LIN {X 0,Y 324.225,Z 783.295,A -85,B 0,C 180,E1 -16076.863,E2 -16076.863} C_VEL
LIN {X 0,Y 323.247,Z 797.636,A -85,B 0,C 180,E1 -16077.399,E2 -16077.399} C_VEL
LIN {X 0,Y 321.791,Z 812,A -85,B 0,C 180,E1 -16078.204,E2 -16078.204} C_VEL
LIN {X 0,Y 320.242,Z 823.952,A -85,B 0,C 180,E1 -16079.097,E2 -16079.097} C_VEL
LIN {X 0,Y 318.471,Z 835.826,A -85,B 0,C 180,E1 -16080.229,E2 -16080.229} C_VEL
LIN {X 0,Y 316.384,Z 847.778,A -85,B 0,C 180,E1 -16081.653,E2 -16081.653} C_VEL
LIN {X 0,Y 314.455,Z 857.682,A -85,B 0,C 180,E1 -16083.091,E2 -16083.091} C_VEL
LIN {X 0,Y 312.599,Z 866.939,A -85,B 0,C 180,E1 -16084.712,E2 -16084.712} C_VEL
LIN {X 0,Y 310.516,Z 876.173,A -85,B 0,C 180,E1 -16086.667,E2 -16086.667} C_VEL
LIN {X 0,Y 308.761,Z 883.843,A -85,B 0,C 180,E1 -16088.642,E2 -16088.642} C_VEL
LIN {X 0,Y 307.38,Z 890.201,A -85,B 0,C 180,E1 -16090.638,E2 -16090.638} C_VEL
LIN {X 0,Y 306.143,Z 895.408,A -85,B 0,C 180,E1 -16092.636,E2 -16092.636} C_VEL
LIN {X 0,Y 305.046,Z 900.883,A -85,B 0,C 180,E1 -16095.319,E2 -16095.319} C_VEL
LIN {X 0,Y 304.213,Z 904.768,A -85,B 0,C 180,E1 -16098,E2 -16098} C_VEL
LIN {X 0,Y 303.829,Z 907.205,A -85,B 0,C 180,E1 -16100.682,E2 -16100.682} C_VEL
LIN {X 0,Y 303.712,Z 908.297,A -85,B 0,C 180,E1 -16103.356,E2 -16103.356} C_VEL
LIN {X 0,Y 303.689,Z 908.077,A -85,B 0,C 180,E1 -16106.019,E2 -16106.019} C_VEL
LIN {X 0,Y 303.703,Z 906.551,A -85,B 0,C 180,E1 -16108.674,E2 -16108.674} C_VEL
LIN {X 0,Y 303.964,Z 903.684,A -85,B 0,C 180,E1 -16111.325,E2 -16111.325} C_VEL
LIN {X 0,Y 304.542,Z 899.397,A -85,B 0,C 180,E1 -16113.97,E2 -16113.97} C_VEL
LIN {X 0,Y 305.582,Z 893.552,A -85,B 0,C 180,E1 -16116.603,E2 -16116.603} C_VEL
LIN {X 0,Y 306.398,Z 887.984,A -85,B 0,C 180,E1 -16118.575,E2 -16118.575} C_VEL
LIN {X 0,Y 307.686,Z 880.207,A -85,B 0,C 180,E1 -16120.828,E2 -16120.828} C_VEL
LIN {X 0,Y 309.255,Z 871.807,A -85,B 0,C 180,E1 -16122.802,E2 -16122.802} C_VEL
LIN {X 0,Y 311.105,Z 861.842,A -85,B 0,C 180,E1 -16124.723,E2 -16124.723} C_VEL
LIN {X 0,Y 312.875,Z 850.729,A -85,B 0,C 180,E1 -16126.475,E2 -16126.475} C_VEL
LIN {X 0,Y 314.508,Z 839.68,A -85,B 0,C 180,E1 -16127.894,E2 -16127.894} C_VEL
LIN {X 0,Y 316.077,Z 827.655,A -85,B 0,C 180,E1 -16129.146,E2 -16129.146} C_VEL
LIN {X 0,Y 317.678,Z 814.307,A -85,B 0,C 180,E1 -16130.223,E2 -16130.223} C_VEL
LIN {X 0,Y 318.794,Z 800.403,A -85,B 0,C 180,E1 -16131.077,E2 -16131.077} C_VEL
LIN {X 0,Y 319.652,Z 785.738,A -85,B 0,C 180,E1 -16131.694,E2 -16131.694} C_VEL
LIN {X 0,Y 320.483,Z 760.014,A -85,B 0,C 180,E1 -16132.31,E2 -16132.31} C_VEL
LIN {X 0,Y 322.515,Z 686.456,A -85,B 0,C 180,E1 -16133.928,E2 -16133.928} C_VEL
LIN {X 0,Y 315.088,Z 668.029,A -85,B 0,C 180,E1 -16135.089,E2 -16135.089} C_VEL
LIN {X 0,Y 307.235,Z 651.005,A -85,B 0,C 180,E1 -16136.326,E2 -16136.326} C_VEL
LIN {X 0,Y 305.705,Z 647.706,A -85,B 0,C 180,E1 -16136.607,E2 -16136.607} C_VEL
LIN {X 0,Y 305.453,Z 646.562,A -85,B 0,C 180,E1 -16137.078,E2 -16137.078} C_VEL
LIN {X 0,Y 305.418,Z 646.57,A -85,B 0,C 180,E1 -16140.414,E2 -16140.414} C_VEL
LIN {X 0,Y 305.462,Z 646.561,A -85,B 0,C 180,E1 -16143.462,E2 -16143.462} C_VEL
LIN {X 0,Y 304.856,Z 646.642,A -85,B 0,C 180,E1 -16144.563,E2 -16144.563} C_VEL
LIN {X 0,Y 301.981,Z 646.998,A -85,B 0,C 180,E1 -16146.353,E2 -16146.353} C_VEL
LIN {X 0,Y 299.499,Z 647.302,A -85,B 0,C 180,E1 -16147.806,E2 -16147.806} C_VEL
LIN {X 0,Y 298.433,Z 647.423,A -85,B 0,C 180,E1 -16148.933,E2 -16148.933} C_VEL
LIN {X 0,Y 298.348,Z 647.43,A -85,B 0,C 180,E1 -16149.315,E2 -16149.315} C_VEL
LIN {X 0,Y 298.402,Z 647.438,A -85,B 0,C 180,E1 -16153.103,E2 -16153.103} C_VEL
LIN {X 0,Y 298.373,Z 647.44,A -85,B 0,C 180,E1 -16156.915,E2 -16156.915} C_VEL
LIN {X 0,Y 298.359,Z 647.429,A -85,B 0,C 180,E1 -16161.017,E2 -16161.017} C_VEL
LIN {X 0,Y 298.406,Z 647.416,A -85,B 0,C 180,E1 -16163.928,E2 -16163.928} C_VEL
LIN {X 0,Y 298.395,Z 647.443,A -85,B 0,C 180,E1 -16167.199,E2 -16167.199} C_VEL
LIN {X 0,Y 298.405,Z 647.428,A -85,B 0,C 180,E1 -16170.625,E2 -16170.625} C_VEL
LIN {X 0,Y 298.442,Z 647.424,A -85,B 0,C 180,E1 -16174.92,E2 -16174.92} C_VEL
LIN {X 0,Y 298.405,Z 647.437,A -85,B 0,C 180,E1 -16177.862,E2 -16177.862} C_VEL
LIN {X 0,Y 298.506,Z 647.422,A -85,B 0,C 180,E1 -16180.754,E2 -16180.754} C_VEL
LIN {X 0,Y 298.588,Z 647.412,A -85,B 0,C 180,E1 -16184.994,E2 -16184.994} C_VEL
LIN {X 0,Y 298.586,Z 647.4,A -85,B 0,C 180,E1 -16189.146,E2 -16189.146} C_VEL
LIN {X 0,Y 298.701,Z 647.398,A -85,B 0,C 180,E1 -16191.884,E2 -16191.884} C_VEL
LIN {X 0,Y 298.639,Z 647.406,A -85,B 0,C 180,E1 -16194.598,E2 -16194.598} C_VEL
LIN {X 0,Y 298.922,Z 647.373,A -85,B 0,C 180,E1 -16198.652,E2 -16198.652} C_VEL
LIN {X 0,Y 298.923,Z 647.365,A -85,B 0,C 180,E1 -16201.347,E2 -16201.347} C_VEL
LIN {X 0,Y 298.788,Z 647.387,A -85,B 0,C 180,E1 -16206.754,E2 -16206.754} C_VEL
LIN {X 0,Y 298.638,Z 647.41,A -85,B 0,C 180,E1 -16209.481,E2 -16209.481} C_VEL
LIN {X 0,Y 298.554,Z 647.42,A -85,B 0,C 180,E1 -16213.615,E2 -16213.615} C_VEL
LIN {X 0,Y 298.551,Z 647.417,A -85,B 0,C 180,E1 -16216.408,E2 -16216.408} C_VEL
LIN {X 0,Y 298.512,Z 647.417,A -85,B 0,C 180,E1 -16219.654,E2 -16219.654} C_VEL
LIN {X 0,Y 298.43,Z 647.428,A -85,B 0,C 180,E1 -16223.6,E2 -16223.6} C_VEL
LIN {X 0,Y 298.491,Z 647.423,A -85,B 0,C 180,E1 -16226.574,E2 -16226.574} C_VEL
LIN {X 0,Y 298.422,Z 647.436,A -85,B 0,C 180,E1 -16229.64,E2 -16229.64} C_VEL
LIN {X 0,Y 298.397,Z 647.439,A -85,B 0,C 180,E1 -16232.8,E2 -16232.8} C_VEL
LIN {X 0,Y 298.467,Z 647.429,A -85,B 0,C 180,E1 -16236.812,E2 -16236.812} C_VEL
LIN {X 0,Y 298.42,Z 647.436,A -85,B 0,C 180,E1 -16241.094,E2 -16241.094} C_VEL
LIN {X 0,Y 298.46,Z 647.431,A -85,B 0,C 180,E1 -16243.115,E2 -16243.115} C_VEL
LIN {X 0,Y 298.403,Z 647.429,A -85,B 0,C 180,E1 -16246.92,E2 -16246.92} C_VEL
LIN {X 0,Y 298.416,Z 647.439,A -85,B 0,C 180,E1 -16251.003,E2 -16251.003} C_VEL
LIN {X 0,Y 298.47,Z 647.46,A -85,B 0,C 180,E1 -16252.143,E2 -16252.143} C_VEL
LIN {X 0,Y 301.205,Z 658.566,A -85,B 0,C 180,E1 -16255.596,E2 -16255.596} C_VEL
LIN {X 0,Y 303.172,Z 667.328,A -85,B 0,C 180,E1 -16258.169,E2 -16258.169} C_VEL
LIN {X 0,Y 310.639,Z 685.569,A -85,B 0,C 180,E1 -16259.416,E2 -16259.416} C_VEL
LIN {X 0,Y 314.632,Z 710.905,A -85,B 0,C 180,E1 -16260.445,E2 -16260.445} C_VEL
LIN {X 0,Y 315.552,Z 718.211,A -85,B 0,C 180,E1 -16260.714,E2 -16260.714} C_VEL
LIN {X 0,Y 313.023,Z 805.174,A -85,B 0,C 180,E1 -16262.686,E2 -16262.686} C_VEL
LIN {X 0,Y 311.976,Z 819.378,A -85,B 0,C 180,E1 -16263.221,E2 -16263.221} C_VEL
LIN {X 0,Y 310.677,Z 833.152,A -85,B 0,C 180,E1 -16264.005,E2 -16264.005} C_VEL
LIN {X 0,Y 309.162,Z 845.617,A -85,B 0,C 180,E1 -16264.951,E2 -16264.951} C_VEL
LIN {X 0,Y 307.467,Z 857.573,A -85,B 0,C 180,E1 -16266.108,E2 -16266.108} C_VEL
LIN {X 0,Y 305.661,Z 869.302,A -85,B 0,C 180,E1 -16267.526,E2 -16267.526} C_VEL
LIN {X 0,Y 303.892,Z 879.332,A -85,B 0,C 180,E1 -16268.994,E2 -16268.994} C_VEL
LIN {X 0,Y 302.222,Z 888.717,A -85,B 0,C 180,E1 -16270.648,E2 -16270.648} C_VEL
LIN {X 0,Y 300.501,Z 898.114,A -85,B 0,C 180,E1 -16272.651,E2 -16272.651} C_VEL
LIN {X 0,Y 299.305,Z 905.27,A -85,B 0,C 180,E1 -16274.493,E2 -16274.493} C_VEL
LIN {X 0,Y 298.259,Z 912.434,A -85,B 0,C 180,E1 -16276.718,E2 -16276.718} C_VEL
LIN {X 0,Y 297.296,Z 918.614,A -85,B 0,C 180,E1 -16279.099,E2 -16279.099} C_VEL
LIN {X 0,Y 296.88,Z 922.825,A -85,B 0,C 180,E1 -16281.148,E2 -16281.148} C_VEL
LIN {X 0,Y 296.684,Z 926.174,A -85,B 0,C 180,E1 -16283.198,E2 -16283.198} C_VEL
LIN {X 0,Y 296.573,Z 929.302,A -85,B 0,C 180,E1 -16285.923,E2 -16285.923} C_VEL
LIN {X 0,Y 296.544,Z 931.034,A -85,B 0,C 180,E1 -16288.642,E2 -16288.642} C_VEL
LIN {X 0,Y 296.581,Z 931.393,A -85,B 0,C 180,E1 -16290,E2 -16290} C_VEL
LIN {X 0,Y 296.545,Z 931.098,A -85,B 0,C 180,E1 -16292.717,E2 -16292.717} C_VEL
LIN {X 0,Y 296.622,Z 929.276,A -85,B 0,C 180,E1 -16295.661,E2 -16295.661} C_VEL
LIN {X 0,Y 296.818,Z 926.457,A -85,B 0,C 180,E1 -16298.167,E2 -16298.167} C_VEL
LIN {X 0,Y 297.389,Z 922.006,A -85,B 0,C 180,E1 -16300.898,E2 -16300.898} C_VEL
LIN {X 0,Y 298.591,Z 915.987,A -85,B 0,C 180,E1 -16303.613,E2 -16303.613} C_VEL
LIN {X 0,Y 300.043,Z 909.183,A -85,B 0,C 180,E1 -16305.991,E2 -16305.991} C_VEL
LIN {X 0,Y 301.762,Z 900.853,A -85,B 0,C 180,E1 -16308.325,E2 -16308.325} C_VEL
LIN {X 0,Y 303.736,Z 892.146,A -85,B 0,C 180,E1 -16310.309,E2 -16310.309} C_VEL
LIN {X 0,Y 306.122,Z 881.619,A -85,B 0,C 180,E1 -16312.26,E2 -16312.26} C_VEL
LIN {X 0,Y 308.672,Z 869.857,A -85,B 0,C 180,E1 -16314.016,E2 -16314.016} C_VEL
LIN {X 0,Y 310.843,Z 858.087,A -85,B 0,C 180,E1 -16315.441,E2 -16315.441} C_VEL
LIN {X 0,Y 312.716,Z 846.881,A -85,B 0,C 180,E1 -16316.53,E2 -16316.53} C_VEL
LIN {X 0,Y 314.636,Z 833.843,A -85,B 0,C 180,E1 -16317.522,E2 -16317.522} C_VEL
LIN {X 0,Y 316.173,Z 821.321,A -85,B 0,C 180,E1 -16318.232,E2 -16318.232} C_VEL
LIN {X 0,Y 317.308,Z 807.323,A -85,B 0,C 180,E1 -16318.799,E2 -16318.799} C_VEL
LIN {X 0,Y 318.368,Z 779.879,A -85,B 0,C 180,E1 -16319.456,E2 -16319.456} C_VEL
LIN {X 0,Y 320.304,Z 717.671,A -85,B 0,C 180,E1 -16320.856,E2 -16320.856} C_VEL
LIN {X 0,Y 316.05,Z 693.353,A -85,B 0,C 180,E1 -16322.001,E2 -16322.001} C_VEL
LIN {X 0,Y 309.511,Z 678.866,A -85,B 0,C 180,E1 -16323.217,E2 -16323.217} C_VEL
LIN {X 0,Y 303.624,Z 666.683,A -85,B 0,C 180,E1 -16324.378,E2 -16324.378} C_VEL
LIN {X 0,Y 301.159,Z 657.209,A -85,B 0,C 180,E1 -16327.492,E2 -16327.492} C_VEL
LIN {X 0,Y 298.416,Z 647.429,A -85,B 0,C 180,E1 -16330.982,E2 -16330.982} C_VEL
LIN {X 0,Y 298.425,Z 647.427,A -85,B 0,C 180,E1 -16333.109,E2 -16333.109} C_VEL
LIN {X 0,Y 298.431,Z 647.424,A -85,B 0,C 180,E1 -16336.926,E2 -16336.926} C_VEL
LIN {X 0,Y 298.425,Z 647.431,A -85,B 0,C 180,E1 -16341.001,E2 -16341.001} C_VEL
LIN {X 0,Y 298.432,Z 647.421,A -85,B 0,C 180,E1 -16343.932,E2 -16343.932} C_VEL
LIN {X 0,Y 298.395,Z 647.411,A -85,B 0,C 180,E1 -16347.983,E2 -16347.983} C_VEL
LIN {X 0,Y 298.464,Z 647.432,A -85,B 0,C 180,E1 -16351.905,E2 -16351.905} C_VEL
LIN {X 0,Y 298.486,Z 647.425,A -85,B 0,C 180,E1 -16354.924,E2 -16354.924} C_VEL
LIN {X 0,Y 298.451,Z 647.432,A -85,B 0,C 180,E1 -16359.316,E2 -16359.316} C_VEL
LIN {X 0,Y 298.539,Z 647.414,A -85,B 0,C 180,E1 -16362.18,E2 -16362.18} C_VEL
LIN {X 0,Y 298.594,Z 647.412,A -85,B 0,C 180,E1 -16364.995,E2 -16364.995} C_VEL
LIN {X 0,Y 298.593,Z 647.414,A -85,B 0,C 180,E1 -16369.147,E2 -16369.147} C_VEL
LIN {X 0,Y 298.742,Z 647.389,A -85,B 0,C 180,E1 -16371.886,E2 -16371.886} C_VEL
LIN {X 0,Y 298.658,Z 647.401,A -85,B 0,C 180,E1 -16374.599,E2 -16374.599} C_VEL
LIN {X 0,Y 298.923,Z 647.374,A -85,B 0,C 180,E1 -16378.653,E2 -16378.653} C_VEL
LIN {X 0,Y 298.923,Z 647.366,A -85,B 0,C 180,E1 -16381.348,E2 -16381.348} C_VEL
LIN {X 0,Y 298.789,Z 647.386,A -85,B 0,C 180,E1 -16386.755,E2 -16386.755} C_VEL
LIN {X 0,Y 298.637,Z 647.405,A -85,B 0,C 180,E1 -16389.482,E2 -16389.482} C_VEL
LIN {X 0,Y 298.554,Z 647.418,A -85,B 0,C 180,E1 -16393.616,E2 -16393.616} C_VEL
LIN {X 0,Y 298.551,Z 647.417,A -85,B 0,C 180,E1 -16396.409,E2 -16396.409} C_VEL
LIN {X 0,Y 298.499,Z 647.418,A -85,B 0,C 180,E1 -16399.648,E2 -16399.648} C_VEL
LIN {X 0,Y 298.425,Z 647.427,A -85,B 0,C 180,E1 -16403.601,E2 -16403.601} C_VEL
LIN {X 0,Y 298.414,Z 647.433,A -85,B 0,C 180,E1 -16406.582,E2 -16406.582} C_VEL
LIN {X 0,Y 298.399,Z 647.411,A -85,B 0,C 180,E1 -16409.644,E2 -16409.644} C_VEL
LIN {X 0,Y 298.394,Z 647.442,A -85,B 0,C 180,E1 -16412.801,E2 -16412.801} C_VEL
LIN {X 0,Y 298.43,Z 647.432,A -85,B 0,C 180,E1 -16416.803,E2 -16416.803} C_VEL
LIN {X 0,Y 298.375,Z 647.435,A -85,B 0,C 180,E1 -16419.492,E2 -16419.492} C_VEL
LIN {X 0,Y 298.401,Z 647.443,A -85,B 0,C 180,E1 -16423.104,E2 -16423.104} C_VEL
LIN {X 0,Y 298.373,Z 647.445,A -85,B 0,C 180,E1 -16426.915,E2 -16426.915} C_VEL
LIN {X 0,Y 298.393,Z 647.622,A -85,B 0,C 180,E1 -16429.581,E2 -16429.581} C_VEL
LIN {X 0,Y 298.698,Z 648.824,A -85,B 0,C 180,E1 -16430.006,E2 -16430.006} C_VEL
LIN {X 0,Y 308.386,Z 665.956,A -85,B 0,C 180,E1 -16431.853,E2 -16431.853} C_VEL
LIN {X 0,Y 316.216,Z 681.809,A -85,B 0,C 180,E1 -16433.288,E2 -16433.288} C_VEL
LIN {X 0,Y 321.076,Z 692.716,A -85,B 0,C 180,E1 -16434.159,E2 -16434.159} C_VEL
LIN {X 0,Y 318.105,Z 784.085,A -85,B 0,C 180,E1 -16436.235,E2 -16436.235} C_VEL
LIN {X 0,Y 317.087,Z 798.194,A -85,B 0,C 180,E1 -16436.779,E2 -16436.779} C_VEL
LIN {X 0,Y 315.58,Z 812.483,A -85,B 0,C 180,E1 -16437.597,E2 -16437.597} C_VEL
LIN {X 0,Y 313.967,Z 824.361,A -85,B 0,C 180,E1 -16438.501,E2 -16438.501} C_VEL
LIN {X 0,Y 311.997,Z 836.946,A -85,B 0,C 180,E1 -16439.734,E2 -16439.734} C_VEL
LIN {X 0,Y 309.843,Z 848.746,A -85,B 0,C 180,E1 -16441.184,E2 -16441.184} C_VEL
LIN {X 0,Y 307.635,Z 859.512,A -85,B 0,C 180,E1 -16442.812,E2 -16442.812} C_VEL
LIN {X 0,Y 305.341,Z 870.141,A -85,B 0,C 180,E1 -16444.798,E2 -16444.798} C_VEL
LIN {X 0,Y 303.243,Z 878.881,A -85,B 0,C 180,E1 -16446.797,E2 -16446.797} C_VEL
LIN {X 0,Y 301.287,Z 886.951,A -85,B 0,C 180,E1 -16449.07,E2 -16449.07} C_VEL
LIN {X 0,Y 299.673,Z 893.906,A -85,B 0,C 180,E1 -16451.542,E2 -16451.542} C_VEL
LIN {X 0,Y 298.323,Z 899.794,A -85,B 0,C 180,E1 -16454.281,E2 -16454.281} C_VEL
LIN {X 0,Y 297.578,Z 903.189,A -85,B 0,C 180,E1 -16456.339,E2 -16456.339} C_VEL
LIN {X 0,Y 296.9,Z 906.377,A -85,B 0,C 180,E1 -16459.084,E2 -16459.084} C_VEL
LIN {X 0,Y 296.682,Z 908.165,A -85,B 0,C 180,E1 -16461.829,E2 -16461.829} C_VEL
LIN {X 0,Y 296.623,Z 908.631,A -85,B 0,C 180,E1 -16464.562,E2 -16464.562} C_VEL
LIN {X 0,Y 296.604,Z 907.792,A -85,B 0,C 180,E1 -16467.284,E2 -16467.284} C_VEL
LIN {X 0,Y 296.718,Z 905.636,A -85,B 0,C 180,E1 -16470,E2 -16470} C_VEL
LIN {X 0,Y 297.101,Z 902.109,A -85,B 0,C 180,E1 -16472.712,E2 -16472.712} C_VEL
LIN {X 0,Y 297.822,Z 898.501,A -85,B 0,C 180,E1 -16474.738,E2 -16474.738} C_VEL
LIN {X 0,Y 298.818,Z 892.248,A -85,B 0,C 180,E1 -16477.433,E2 -16477.433} C_VEL
LIN {X 0,Y 299.862,Z 886.39,A -85,B 0,C 180,E1 -16479.443,E2 -16479.443} C_VEL
LIN {X 0,Y 301.192,Z 878.162,A -85,B 0,C 180,E1 -16481.747,E2 -16481.747} C_VEL
LIN {X 0,Y 302.992,Z 869.277,A -85,B 0,C 180,E1 -16483.754,E2 -16483.754} C_VEL
LIN {X 0,Y 304.932,Z 858.691,A -85,B 0,C 180,E1 -16485.713,E2 -16485.713} C_VEL
LIN {X 0,Y 306.708,Z 847.993,A -85,B 0,C 180,E1 -16487.331,E2 -16487.331} C_VEL
LIN {X 0,Y 308.334,Z 836.313,A -85,B 0,C 180,E1 -16488.782,E2 -16488.782} C_VEL
LIN {X 0,Y 310.134,Z 823.398,A -85,B 0,C 180,E1 -16490.045,E2 -16490.045} C_VEL
LIN {X 0,Y 311.63,Z 809.884,A -85,B 0,C 180,E1 -16491.065,E2 -16491.065} C_VEL
LIN {X 0,Y 312.735,Z 795.632,A -85,B 0,C 180,E1 -16491.852,E2 -16491.852} C_VEL
LIN {X 0,Y 313.458,Z 781.713,A -85,B 0,C 180,E1 -16492.362,E2 -16492.362} C_VEL
LIN {X 0,Y 316.225,Z 688.388,A -85,B 0,C 180,E1 -16494.465,E2 -16494.465} C_VEL
LIN {X 0,Y 308.861,Z 670.042,A -85,B 0,C 180,E1 -16495.659,E2 -16495.659} C_VEL
LIN {X 0,Y 300.183,Z 651.551,A -85,B 0,C 180,E1 -16497.075,E2 -16497.075} C_VEL
LIN {X 0,Y 298.544,Z 648.169,A -85,B 0,C 180,E1 -16497.351,E2 -16497.351} C_VEL
LIN {X 0,Y 298.402,Z 647.444,A -85,B 0,C 180,E1 -16497.637,E2 -16497.637} C_VEL
LIN {X 0,Y 298.39,Z 647.443,A -85,B 0,C 180,E1 -16502.014,E2 -16502.014} C_VEL
LIN {X 0,Y 298.432,Z 647.435,A -85,B 0,C 180,E1 -16504.487,E2 -16504.487} C_VEL
LIN {X 0,Y 298.389,Z 647.441,A -85,B 0,C 180,E1 -16507.762,E2 -16507.762} C_VEL
LIN {X 0,Y 298.348,Z 647.43,A -85,B 0,C 180,E1 -16509.315,E2 -16509.315} C_VEL
LIN {X 0,Y 297.68,Z 647.514,A -85,B 0,C 180,E1 -16510.442,E2 -16510.442} C_VEL
LIN {X 0,Y 294.805,Z 647.887,A -85,B 0,C 180,E1 -16512.276,E2 -16512.276} C_VEL
LIN {X 0,Y 292.376,Z 648.187,A -85,B 0,C 180,E1 -16513.765,E2 -16513.765} C_VEL
LIN {X 0,Y 291.35,Z 648.316,A -85,B 0,C 180,E1 -16514.919,E2 -16514.919} C_VEL
LIN {X 0,Y 291.275,Z 648.325,A -85,B 0,C 180,E1 -16515.309,E2 -16515.309} C_VEL
LIN {X 0,Y 291.297,Z 648.324,A -85,B 0,C 180,E1 -16519.351,E2 -16519.351} C_VEL
LIN {X 0,Y 291.389,Z 648.282,A -85,B 0,C 180,E1 -16522.916,E2 -16522.916} C_VEL
LIN {X 0,Y 291.346,Z 648.316,A -85,B 0,C 180,E1 -16526.301,E2 -16526.301} C_VEL
LIN {X 0,Y 291.368,Z 648.303,A -85,B 0,C 180,E1 -16530.268,E2 -16530.268} C_VEL
LIN {X 0,Y 291.361,Z 648.311,A -85,B 0,C 180,E1 -16534.266,E2 -16534.266} C_VEL
LIN {X 0,Y 291.367,Z 648.306,A -85,B 0,C 180,E1 -16537.298,E2 -16537.298} C_VEL
LIN {X 0,Y 291.442,Z 648.302,A -85,B 0,C 180,E1 -16540.269,E2 -16540.269} C_VEL
LIN {X 0,Y 291.517,Z 648.292,A -85,B 0,C 180,E1 -16544.653,E2 -16544.653} C_VEL
LIN {X 0,Y 291.532,Z 648.279,A -85,B 0,C 180,E1 -16548.88,E2 -16548.88} C_VEL
LIN {X 0,Y 291.654,Z 648.273,A -85,B 0,C 180,E1 -16551.686,E2 -16551.686} C_VEL
LIN {X 0,Y 291.608,Z 648.282,A -85,B 0,C 180,E1 -16554.467,E2 -16554.467} C_VEL
LIN {X 0,Y 291.889,Z 648.249,A -85,B 0,C 180,E1 -16558.62,E2 -16558.62} C_VEL
LIN {X 0,Y 291.889,Z 648.241,A -85,B 0,C 180,E1 -16561.379,E2 -16561.379} C_VEL
LIN {X 0,Y 291.737,Z 648.265,A -85,B 0,C 180,E1 -16566.918,E2 -16566.918} C_VEL
LIN {X 0,Y 291.577,Z 648.286,A -85,B 0,C 180,E1 -16569.713,E2 -16569.713} C_VEL
LIN {X 0,Y 291.524,Z 648.294,A -85,B 0,C 180,E1 -16573.95,E2 -16573.95} C_VEL
LIN {X 0,Y 291.489,Z 648.297,A -85,B 0,C 180,E1 -16576.817,E2 -16576.817} C_VEL
LIN {X 0,Y 291.452,Z 648.297,A -85,B 0,C 180,E1 -16579.874,E2 -16579.874} C_VEL
LIN {X 0,Y 291.384,Z 648.307,A -85,B 0,C 180,E1 -16584.206,E2 -16584.206} C_VEL
LIN {X 0,Y 291.424,Z 648.301,A -85,B 0,C 180,E1 -16587.271,E2 -16587.271} C_VEL
LIN {X 0,Y 291.339,Z 648.315,A -85,B 0,C 180,E1 -16590.436,E2 -16590.436} C_VEL
LIN {X 0,Y 291.346,Z 648.316,A -85,B 0,C 180,E1 -16593.698,E2 -16593.698} C_VEL
LIN {X 0,Y 291.402,Z 648.31,A -85,B 0,C 180,E1 -16597.26,E2 -16597.26} C_VEL
LIN {X 0,Y 291.379,Z 648.316,A -85,B 0,C 180,E1 -16600.634,E2 -16600.634} C_VEL
LIN {X 0,Y 291.333,Z 648.318,A -85,B 0,C 180,E1 -16604.393,E2 -16604.393} C_VEL
LIN {X 0,Y 291.328,Z 648.321,A -85,B 0,C 180,E1 -16608.404,E2 -16608.404} C_VEL
LIN {X 0,Y 291.439,Z 648.509,A -85,B 0,C 180,E1 -16611.543,E2 -16611.543} C_VEL
LIN {X 0,Y 294.13,Z 659.279,A -85,B 0,C 180,E1 -16615.008,E2 -16615.008} C_VEL
LIN {X 0,Y 295.851,Z 666.97,A -85,B 0,C 180,E1 -16617.347,E2 -16617.347} C_VEL
LIN {X 0,Y 304.416,Z 687.348,A -85,B 0,C 180,E1 -16618.832,E2 -16618.832} C_VEL
LIN {X 0,Y 307.154,Z 703.717,A -85,B 0,C 180,E1 -16619.539,E2 -16619.539} C_VEL
LIN {X 0,Y 309.223,Z 719.038,A -85,B 0,C 180,E1 -16620.138,E2 -16620.138} C_VEL
LIN {X 0,Y 306.575,Z 805.95,A -85,B 0,C 180,E1 -16622.155,E2 -16622.155} C_VEL
LIN {X 0,Y 305.41,Z 820.519,A -85,B 0,C 180,E1 -16622.737,E2 -16622.737} C_VEL
LIN {X 0,Y 304.155,Z 833.362,A -85,B 0,C 180,E1 -16623.497,E2 -16623.497} C_VEL
LIN {X 0,Y 302.452,Z 846.611,A -85,B 0,C 180,E1 -16624.54,E2 -16624.54} C_VEL
LIN {X 0,Y 300.52,Z 859.533,A -85,B 0,C 180,E1 -16625.858,E2 -16625.858} C_VEL
LIN {X 0,Y 298.669,Z 871.063,A -85,B 0,C 180,E1 -16627.336,E2 -16627.336} C_VEL
LIN {X 0,Y 296.806,Z 880.745,A -85,B 0,C 180,E1 -16628.832,E2 -16628.832} C_VEL
LIN {X 0,Y 294.836,Z 891.508,A -85,B 0,C 180,E1 -16630.867,E2 -16630.867} C_VEL
LIN {X 0,Y 293.14,Z 900.385,A -85,B 0,C 180,E1 -16632.921,E2 -16632.921} C_VEL
LIN {X 0,Y 292.024,Z 907.781,A -85,B 0,C 180,E1 -16635.006,E2 -16635.006} C_VEL
LIN {X 0,Y 290.821,Z 914.841,A -85,B 0,C 180,E1 -16637.438,E2 -16637.438} C_VEL
LIN {X 0,Y 290.094,Z 919.733,A -85,B 0,C 180,E1 -16639.531,E2 -16639.531} C_VEL
LIN {X 0,Y 289.654,Z 924.792,A -85,B 0,C 180,E1 -16642.331,E2 -16642.331} C_VEL
LIN {X 0,Y 289.515,Z 927.59,A -85,B 0,C 180,E1 -16644.428,E2 -16644.428} C_VEL
LIN {X 0,Y 289.486,Z 930.038,A -85,B 0,C 180,E1 -16647.217,E2 -16647.217} C_VEL
LIN {X 0,Y 289.496,Z 931.115,A -85,B 0,C 180,E1 -16650,E2 -16650} C_VEL
LIN {X 0,Y 289.471,Z 930.842,A -85,B 0,C 180,E1 -16652.783,E2 -16652.783} C_VEL
LIN {X 0,Y 289.515,Z 929.228,A -85,B 0,C 180,E1 -16655.572,E2 -16655.572} C_VEL
LIN {X 0,Y 289.754,Z 926.246,A -85,B 0,C 180,E1 -16658.368,E2 -16658.368} C_VEL
LIN {X 0,Y 290.357,Z 921.819,A -85,B 0,C 180,E1 -16661.165,E2 -16661.165} C_VEL
LIN {X 0,Y 291.637,Z 915.832,A -85,B 0,C 180,E1 -16663.945,E2 -16663.945} C_VEL
LIN {X 0,Y 293.185,Z 908.693,A -85,B 0,C 180,E1 -16666.495,E2 -16666.495} C_VEL
LIN {X 0,Y 294.988,Z 900.771,A -85,B 0,C 180,E1 -16668.762,E2 -16668.762} C_VEL
LIN {X 0,Y 297.056,Z 892.106,A -85,B 0,C 180,E1 -16670.786,E2 -16670.786} C_VEL
LIN {X 0,Y 299.564,Z 881.627,A -85,B 0,C 180,E1 -16672.774,E2 -16672.774} C_VEL
LIN {X 0,Y 302.186,Z 869.924,A -85,B 0,C 180,E1 -16674.565,E2 -16674.565} C_VEL
LIN {X 0,Y 304.452,Z 858.227,A -85,B 0,C 180,E1 -16676.014,E2 -16676.014} C_VEL
LIN {X 0,Y 306.677,Z 845.358,A -85,B 0,C 180,E1 -16677.279,E2 -16677.279} C_VEL
LIN {X 0,Y 308.729,Z 831.97,A -85,B 0,C 180,E1 -16678.28,E2 -16678.28} C_VEL
LIN {X 0,Y 310.214,Z 819.654,A -85,B 0,C 180,E1 -16678.964,E2 -16678.964} C_VEL
LIN {X 0,Y 311.332,Z 806.097,A -85,B 0,C 180,E1 -16679.498,E2 -16679.498} C_VEL
LIN {X 0,Y 313.639,Z 740.667,A -85,B 0,C 180,E1 -16681.023,E2 -16681.023} C_VEL
LIN {X 0,Y 314.282,Z 718.374,A -85,B 0,C 180,E1 -16681.543,E2 -16681.543} C_VEL
LIN {X 0,Y 310.455,Z 696.266,A -85,B 0,C 180,E1 -16682.615,E2 -16682.615} C_VEL
LIN {X 0,Y 304.115,Z 682.195,A -85,B 0,C 180,E1 -16683.839,E2 -16683.839} C_VEL
LIN {X 0,Y 296.363,Z 666.32,A -85,B 0,C 180,E1 -16685.429,E2 -16685.429} C_VEL
LIN {X 0,Y 293.326,Z 655.076,A -85,B 0,C 180,E1 -16689.327,E2 -16689.327} C_VEL
LIN {X 0,Y 291.359,Z 648.316,A -85,B 0,C 180,E1 -16691.854,E2 -16691.854} C_VEL
LIN {X 0,Y 291.323,Z 648.322,A -85,B 0,C 180,E1 -16695.605,E2 -16695.605} C_VEL
LIN {X 0,Y 291.376,Z 648.309,A -85,B 0,C 180,E1 -16699.365,E2 -16699.365} C_VEL
LIN {X 0,Y 291.428,Z 648.286,A -85,B 0,C 180,E1 -16702.923,E2 -16702.923} C_VEL
LIN {X 0,Y 291.345,Z 648.314,A -85,B 0,C 180,E1 -16706.302,E2 -16706.302} C_VEL
LIN {X 0,Y 291.387,Z 648.296,A -85,B 0,C 180,E1 -16710.26,E2 -16710.26} C_VEL
LIN {X 0,Y 291.417,Z 648.302,A -85,B 0,C 180,E1 -16714.272,E2 -16714.272} C_VEL
LIN {X 0,Y 291.382,Z 648.305,A -85,B 0,C 180,E1 -16717.3,E2 -16717.3} C_VEL
LIN {X 0,Y 291.459,Z 648.302,A -85,B 0,C 180,E1 -16720.271,E2 -16720.271} C_VEL
LIN {X 0,Y 291.556,Z 648.29,A -85,B 0,C 180,E1 -16724.624,E2 -16724.624} C_VEL
LIN {X 0,Y 291.537,Z 648.294,A -85,B 0,C 180,E1 -16728.881,E2 -16728.881} C_VEL
LIN {X 0,Y 291.688,Z 648.266,A -85,B 0,C 180,E1 -16731.688,E2 -16731.688} C_VEL
LIN {X 0,Y 291.628,Z 648.277,A -85,B 0,C 180,E1 -16734.469,E2 -16734.469} C_VEL
LIN {X 0,Y 291.89,Z 648.25,A -85,B 0,C 180,E1 -16738.621,E2 -16738.621} C_VEL
LIN {X 0,Y 291.89,Z 648.242,A -85,B 0,C 180,E1 -16741.38,E2 -16741.38} C_VEL
LIN {X 0,Y 291.737,Z 648.266,A -85,B 0,C 180,E1 -16746.919,E2 -16746.919} C_VEL
LIN {X 0,Y 291.577,Z 648.282,A -85,B 0,C 180,E1 -16749.714,E2 -16749.714} C_VEL
LIN {X 0,Y 291.524,Z 648.293,A -85,B 0,C 180,E1 -16753.951,E2 -16753.951} C_VEL
LIN {X 0,Y 291.488,Z 648.301,A -85,B 0,C 180,E1 -16756.818,E2 -16756.818} C_VEL
LIN {X 0,Y 291.452,Z 648.296,A -85,B 0,C 180,E1 -16759.875,E2 -16759.875} C_VEL
LIN {X 0,Y 291.366,Z 648.309,A -85,B 0,C 180,E1 -16764.209,E2 -16764.209} C_VEL
LIN {X 0,Y 291.36,Z 648.303,A -85,B 0,C 180,E1 -16767.278,E2 -16767.278} C_VEL
LIN {X 0,Y 291.322,Z 648.3,A -85,B 0,C 180,E1 -16770.439,E2 -16770.439} C_VEL
LIN {X 0,Y 291.345,Z 648.312,A -85,B 0,C 180,E1 -16773.699,E2 -16773.699} C_VEL
LIN {X 0,Y 291.361,Z 648.313,A -85,B 0,C 180,E1 -16777.25,E2 -16777.25} C_VEL
LIN {X 0,Y 291.301,Z 648.305,A -85,B 0,C 180,E1 -16780.649,E2 -16780.649} C_VEL
LIN {X 0,Y 291.292,Z 648.319,A -85,B 0,C 180,E1 -16784.402,E2 -16784.402} C_VEL
LIN {X 0,Y 291.326,Z 648.339,A -85,B 0,C 180,E1 -16788.642,E2 -16788.642} C_VEL
LIN {X 0,Y 291.428,Z 649.017,A -85,B 0,C 180,E1 -16788.904,E2 -16788.904} C_VEL
LIN {X 0,Y 292.744,Z 651.781,A -85,B 0,C 180,E1 -16789.198,E2 -16789.198} C_VEL
LIN {X 0,Y 294.482,Z 654.35,A -85,B 0,C 180,E1 -16789.543,E2 -16789.543} C_VEL
LIN {X 0,Y 301.594,Z 666.811,A -85,B 0,C 180,E1 -16790.95,E2 -16790.95} C_VEL
LIN {X 0,Y 308.318,Z 679.777,A -85,B 0,C 180,E1 -16792.231,E2 -16792.231} C_VEL
LIN {X 0,Y 315.092,Z 694.702,A -85,B 0,C 180,E1 -16793.497,E2 -16793.497} C_VEL
LIN {X 0,Y 312,Z 785.032,A -85,B 0,C 180,E1 -16795.59,E2 -16795.59} C_VEL
LIN {X 0,Y 310.88,Z 799.519,A -85,B 0,C 180,E1 -16796.173,E2 -16796.173} C_VEL
LIN {X 0,Y 309.417,Z 812.968,A -85,B 0,C 180,E1 -16796.967,E2 -16796.967} C_VEL
LIN {X 0,Y 307.877,Z 823.87,A -85,B 0,C 180,E1 -16797.799,E2 -16797.799} C_VEL
LIN {X 0,Y 305.819,Z 836.634,A -85,B 0,C 180,E1 -16799.056,E2 -16799.056} C_VEL
LIN {X 0,Y 303.556,Z 848.538,A -85,B 0,C 180,E1 -16800.529,E2 -16800.529} C_VEL
LIN {X 0,Y 301.246,Z 859.385,A -85,B 0,C 180,E1 -16802.187,E2 -16802.187} C_VEL
LIN {X 0,Y 298.849,Z 870.082,A -85,B 0,C 180,E1 -16804.211,E2 -16804.211} C_VEL
LIN {X 0,Y 296.653,Z 878.876,A -85,B 0,C 180,E1 -16806.25,E2 -16806.25} C_VEL
LIN {X 0,Y 294.677,Z 886.633,A -85,B 0,C 180,E1 -16808.459,E2 -16808.459} C_VEL
LIN {X 0,Y 292.836,Z 894.006,A -85,B 0,C 180,E1 -16811.095,E2 -16811.095} C_VEL
LIN {X 0,Y 291.391,Z 899.941,A -85,B 0,C 180,E1 -16813.897,E2 -16813.897} C_VEL
LIN {X 0,Y 290.605,Z 903.355,A -85,B 0,C 180,E1 -16816.005,E2 -16816.005} C_VEL
LIN {X 0,Y 289.854,Z 906.591,A -85,B 0,C 180,E1 -16818.815,E2 -16818.815} C_VEL
LIN {X 0,Y 289.616,Z 908.415,A -85,B 0,C 180,E1 -16821.628,E2 -16821.628} C_VEL
LIN {X 0,Y 289.559,Z 908.912,A -85,B 0,C 180,E1 -16824.429,E2 -16824.429} C_VEL
LIN {X 0,Y 289.528,Z 908.106,A -85,B 0,C 180,E1 -16827.217,E2 -16827.217} C_VEL
LIN {X 0,Y 289.626,Z 905.984,A -85,B 0,C 180,E1 -16830,E2 -16830} C_VEL
LIN {X 0,Y 290.02,Z 902.491,A -85,B 0,C 180,E1 -16832.778,E2 -16832.778} C_VEL
LIN {X 0,Y 290.767,Z 898.92,A -85,B 0,C 180,E1 -16834.853,E2 -16834.853} C_VEL
LIN {X 0,Y 291.788,Z 892.707,A -85,B 0,C 180,E1 -16837.613,E2 -16837.613} C_VEL
LIN {X 0,Y 293.074,Z 885.7,A -85,B 0,C 180,E1 -16840.041,E2 -16840.041} C_VEL
LIN {X 0,Y 294.524,Z 877.243,A -85,B 0,C 180,E1 -16842.402,E2 -16842.402} C_VEL
LIN {X 0,Y 296.454,Z 868.272,A -85,B 0,C 180,E1 -16844.414,E2 -16844.414} C_VEL
LIN {X 0,Y 298.528,Z 857.428,A -85,B 0,C 180,E1 -16846.41,E2 -16846.41} C_VEL
LIN {X 0,Y 300.424,Z 846.408,A -85,B 0,C 180,E1 -16848.057,E2 -16848.057} C_VEL
LIN {X 0,Y 302.14,Z 834.27,A -85,B 0,C 180,E1 -16849.535,E2 -16849.535} C_VEL
LIN {X 0,Y 303.773,Z 822.598,A -85,B 0,C 180,E1 -16850.66,E2 -16850.66} C_VEL
LIN {X 0,Y 305.277,Z 808.644,A -85,B 0,C 180,E1 -16851.703,E2 -16851.703} C_VEL
LIN {X 0,Y 306.37,Z 794.668,A -85,B 0,C 180,E1 -16852.463,E2 -16852.463} C_VEL
LIN {X 0,Y 307.138,Z 780.5,A -85,B 0,C 180,E1 -16852.965,E2 -16852.965} C_VEL
LIN {X 0,Y 309.867,Z 690.077,A -85,B 0,C 180,E1 -16855.039,E2 -16855.039} C_VEL
LIN {X 0,Y 303.079,Z 673.187,A -85,B 0,C 180,E1 -16856.178,E2 -16856.178} C_VEL
LIN {X 0,Y 295.601,Z 657.05,A -85,B 0,C 180,E1 -16857.441,E2 -16857.441} C_VEL
LIN {X 0,Y 292.562,Z 651.486,A -85,B 0,C 180,E1 -16857.949,E2 -16857.949} C_VEL
LIN {X 0,Y 291.451,Z 648.879,A -85,B 0,C 180,E1 -16858.154,E2 -16858.154} C_VEL
LIN {X 0,Y 291.351,Z 648.317,A -85,B 0,C 180,E1 -16858.251,E2 -16858.251} C_VEL
LIN {X 0,Y 291.34,Z 648.32,A -85,B 0,C 180,E1 -16862.401,E2 -16862.401} C_VEL
LIN {X 0,Y 291.358,Z 648.318,A -85,B 0,C 180,E1 -16865.375,E2 -16865.375} C_VEL
LIN {X 0,Y 291.307,Z 648.311,A -85,B 0,C 180,E1 -16868.849,E2 -16868.849} C_VEL
LIN {X 0,Y 291.316,Z 648.323,A -85,B 0,C 180,E1 -16872.493,E2 -16872.493} C_VEL
LIN {X 0,Y 291.275,Z 648.325,A -85,B 0,C 180,E1 -16875.309,E2 -16875.309} C_VEL
LIN {X 0,Y 290.621,Z 648.412,A -85,B 0,C 180,E1 -16876.462,E2 -16876.462} C_VEL
LIN {X 0,Y 287.745,Z 648.766,A -85,B 0,C 180,E1 -16878.339,E2 -16878.339} C_VEL
LIN {X 0,Y 285.317,Z 649.066,A -85,B 0,C 180,E1 -16879.862,E2 -16879.862} C_VEL
LIN {X 0,Y 284.307,Z 649.177,A -85,B 0,C 180,E1 -16881.044,E2 -16881.044} C_VEL
LIN {X 0,Y 284.243,Z 649.178,A -85,B 0,C 180,E1 -16881.444,E2 -16881.444} C_VEL
LIN {X 0,Y 284.339,Z 649.176,A -85,B 0,C 180,E1 -16884.653,E2 -16884.653} C_VEL
LIN {X 0,Y 284.288,Z 649.19,A -85,B 0,C 180,E1 -16888.724,E2 -16888.724} C_VEL
LIN {X 0,Y 284.286,Z 649.197,A -85,B 0,C 180,E1 -16891.984,E2 -16891.984} C_VEL
LIN {X 0,Y 284.323,Z 649.177,A -85,B 0,C 180,E1 -16896.147,E2 -16896.147} C_VEL
LIN {X 0,Y 284.379,Z 649.183,A -85,B 0,C 180,E1 -16899.904,E2 -16899.904} C_VEL
LIN {X 0,Y 284.457,Z 649.171,A -85,B 0,C 180,E1 -16904.486,E2 -16904.486} C_VEL
LIN {X 0,Y 284.485,Z 649.159,A -85,B 0,C 180,E1 -16908.601,E2 -16908.601} C_VEL
LIN {X 0,Y 284.611,Z 649.148,A -85,B 0,C 180,E1 -16911.479,E2 -16911.479} C_VEL
LIN {X 0,Y 284.577,Z 649.158,A -85,B 0,C 180,E1 -16914.33,E2 -16914.33} C_VEL
LIN {X 0,Y 284.855,Z 649.126,A -85,B 0,C 180,E1 -16918.586,E2 -16918.586} C_VEL
LIN {X 0,Y 284.856,Z 649.118,A -85,B 0,C 180,E1 -16921.413,E2 -16921.413} C_VEL
LIN {X 0,Y 284.688,Z 649.143,A -85,B 0,C 180,E1 -16927.09,E2 -16927.09} C_VEL
LIN {X 0,Y 284.521,Z 649.162,A -85,B 0,C 180,E1 -16929.957,E2 -16929.957} C_VEL
LIN {X 0,Y 284.484,Z 649.167,A -85,B 0,C 180,E1 -16934.302,E2 -16934.302} C_VEL
LIN {X 0,Y 284.428,Z 649.177,A -85,B 0,C 180,E1 -16937.248,E2 -16937.248} C_VEL
LIN {X 0,Y 284.379,Z 649.179,A -85,B 0,C 180,E1 -16940.242,E2 -16940.242} C_VEL
LIN {X 0,Y 284.34,Z 649.189,A -85,B 0,C 180,E1 -16944.846,E2 -16944.846} C_VEL
LIN {X 0,Y 284.333,Z 649.186,A -85,B 0,C 180,E1 -16948.01,E2 -16948.01} C_VEL
LIN {X 0,Y 284.298,Z 649.192,A -85,B 0,C 180,E1 -16951.274,E2 -16951.274} C_VEL
LIN {X 0,Y 284.363,Z 649.188,A -85,B 0,C 180,E1 -16955.354,E2 -16955.354} C_VEL
LIN {X 0,Y 284.334,Z 649.193,A -85,B 0,C 180,E1 -16958.165,E2 -16958.165} C_VEL
LIN {X 0,Y 284.304,Z 649.193,A -85,B 0,C 180,E1 -16961.87,E2 -16961.87} C_VEL
LIN {X 0,Y 284.266,Z 649.195,A -85,B 0,C 180,E1 -16965.805,E2 -16965.805} C_VEL
LIN {X 0,Y 284.307,Z 649.197,A -85,B 0,C 180,E1 -16970.023,E2 -16970.023} C_VEL
LIN {X 0,Y 284.341,Z 649.269,A -85,B 0,C 180,E1 -16970.815,E2 -16970.815} C_VEL
LIN {X 0,Y 286.805,Z 658.691,A -85,B 0,C 180,E1 -16973.977,E2 -16973.977} C_VEL
LIN {X 0,Y 288.662,Z 666.766,A -85,B 0,C 180,E1 -16976.514,E2 -16976.514} C_VEL
LIN {X 0,Y 298.32,Z 689.569,A -85,B 0,C 180,E1 -16978.246,E2 -16978.246} C_VEL
LIN {X 0,Y 299.612,Z 696.343,A -85,B 0,C 180,E1 -16978.567,E2 -16978.567} C_VEL
LIN {X 0,Y 302.925,Z 719.909,A -85,B 0,C 180,E1 -16979.538,E2 -16979.538} C_VEL
LIN {X 0,Y 300.197,Z 805.483,A -85,B 0,C 180,E1 -16981.557,E2 -16981.557} C_VEL
LIN {X 0,Y 299.033,Z 820.122,A -85,B 0,C 180,E1 -16982.153,E2 -16982.153} C_VEL
LIN {X 0,Y 297.632,Z 833.562,A -85,B 0,C 180,E1 -16982.964,E2 -16982.964} C_VEL
LIN {X 0,Y 295.999,Z 845.817,A -85,B 0,C 180,E1 -16983.944,E2 -16983.944} C_VEL
LIN {X 0,Y 294.002,Z 858.796,A -85,B 0,C 180,E1 -16985.281,E2 -16985.281} C_VEL
LIN {X 0,Y 292.068,Z 870.443,A -85,B 0,C 180,E1 -16986.794,E2 -16986.794} C_VEL
LIN {X 0,Y 290.18,Z 880.188,A -85,B 0,C 180,E1 -16988.324,E2 -16988.324} C_VEL
LIN {X 0,Y 288.414,Z 889.351,A -85,B 0,C 180,E1 -16990.053,E2 -16990.053} C_VEL
LIN {X 0,Y 286.571,Z 898.543,A -85,B 0,C 180,E1 -16992.148,E2 -16992.148} C_VEL
LIN {X 0,Y 285.198,Z 906.206,A -85,B 0,C 180,E1 -16994.272,E2 -16994.272} C_VEL
LIN {X 0,Y 284.167,Z 912.6,A -85,B 0,C 180,E1 -16996.411,E2 -16996.411} C_VEL
LIN {X 0,Y 283.067,Z 919.357,A -85,B 0,C 180,E1 -16999.268,E2 -16999.268} C_VEL
LIN {X 0,Y 282.57,Z 924.441,A -85,B 0,C 180,E1 -17002.137,E2 -17002.137} C_VEL
LIN {X 0,Y 282.413,Z 927.497,A -85,B 0,C 180,E1 -17004.513,E2 -17004.513} C_VEL
LIN {X 0,Y 282.413,Z 929.737,A -85,B 0,C 180,E1 -17007.147,E2 -17007.147} C_VEL
LIN {X 0,Y 282.413,Z 930.836,A -85,B 0,C 180,E1 -17010,E2 -17010} C_VEL
LIN {X 0,Y 282.376,Z 930.586,A -85,B 0,C 180,E1 -17012.853,E2 -17012.853} C_VEL
LIN {X 0,Y 282.438,Z 928.994,A -85,B 0,C 180,E1 -17015.712,E2 -17015.712} C_VEL
LIN {X 0,Y 282.683,Z 926.034,A -85,B 0,C 180,E1 -17018.579,E2 -17018.579} C_VEL
LIN {X 0,Y 283.338,Z 921.632,A -85,B 0,C 180,E1 -17021.445,E2 -17021.445} C_VEL
LIN {X 0,Y 284.684,Z 915.675,A -85,B 0,C 180,E1 -17024.292,E2 -17024.292} C_VEL
LIN {X 0,Y 286.226,Z 909.06,A -85,B 0,C 180,E1 -17026.743,E2 -17026.743} C_VEL
LIN {X 0,Y 288.243,Z 900.694,A -85,B 0,C 180,E1 -17029.218,E2 -17029.218} C_VEL
LIN {X 0,Y 290.401,Z 892.068,A -85,B 0,C 180,E1 -17031.285,E2 -17031.285} C_VEL
LIN {X 0,Y 293.026,Z 881.636,A -85,B 0,C 180,E1 -17033.312,E2 -17033.312} C_VEL
LIN {X 0,Y 295.733,Z 869.991,A -85,B 0,C 180,E1 -17035.138,E2 -17035.138} C_VEL
LIN {X 0,Y 298.087,Z 858.368,A -85,B 0,C 180,E1 -17036.613,E2 -17036.613} C_VEL
LIN {X 0,Y 300.395,Z 845.597,A -85,B 0,C 180,E1 -17037.899,E2 -17037.899} C_VEL
LIN {X 0,Y 302.524,Z 832.352,A -85,B 0,C 180,E1 -17038.914,E2 -17038.914} C_VEL
LIN {X 0,Y 304.054,Z 820.263,A -85,B 0,C 180,E1 -17039.608,E2 -17039.608} C_VEL
LIN {X 0,Y 305.191,Z 807.147,A -85,B 0,C 180,E1 -17040.152,E2 -17040.152} C_VEL
LIN {X 0,Y 306.222,Z 783.063,A -85,B 0,C 180,E1 -17040.758,E2 -17040.758} C_VEL
LIN {X 0,Y 308.413,Z 719.928,A -85,B 0,C 180,E1 -17042.221,E2 -17042.221} C_VEL
LIN {X 0,Y 304.853,Z 699.005,A -85,B 0,C 180,E1 -17043.263,E2 -17043.263} C_VEL
LIN {X 0,Y 297.837,Z 683.484,A -85,B 0,C 180,E1 -17044.673,E2 -17044.673} C_VEL
LIN {X 0,Y 291.015,Z 669.953,A -85,B 0,C 180,E1 -17046.089,E2 -17046.089} C_VEL
LIN {X 0,Y 289.042,Z 666.009,A -85,B 0,C 180,E1 -17046.543,E2 -17046.543} C_VEL
LIN {X 0,Y 286.463,Z 656.411,A -85,B 0,C 180,E1 -17050.002,E2 -17050.002} C_VEL
LIN {X 0,Y 284.296,Z 649.189,A -85,B 0,C 180,E1 -17052.863,E2 -17052.863} C_VEL
LIN {X 0,Y 284.286,Z 649.195,A -85,B 0,C 180,E1 -17056.196,E2 -17056.196} C_VEL
LIN {X 0,Y 284.351,Z 649.192,A -85,B 0,C 180,E1 -17060.013,E2 -17060.013} C_VEL
LIN {X 0,Y 284.352,Z 649.171,A -85,B 0,C 180,E1 -17063.617,E2 -17063.617} C_VEL
LIN {X 0,Y 284.308,Z 649.174,A -85,B 0,C 180,E1 -17067.19,E2 -17067.19} C_VEL
LIN {X 0,Y 284.359,Z 649.172,A -85,B 0,C 180,E1 -17070.376,E2 -17070.376} C_VEL
LIN {X 0,Y 284.378,Z 649.177,A -85,B 0,C 180,E1 -17073.587,E2 -17073.587} C_VEL
LIN {X 0,Y 284.367,Z 649.182,A -85,B 0,C 180,E1 -17076.707,E2 -17076.707} C_VEL
LIN {X 0,Y 284.404,Z 649.175,A -85,B 0,C 180,E1 -17081.262,E2 -17081.262} C_VEL
LIN {X 0,Y 284.493,Z 649.171,A -85,B 0,C 180,E1 -17084.459,E2 -17084.459} C_VEL
LIN {X 0,Y 284.488,Z 649.173,A -85,B 0,C 180,E1 -17088.602,E2 -17088.602} C_VEL
LIN {X 0,Y 284.64,Z 649.143,A -85,B 0,C 180,E1 -17091.481,E2 -17091.481} C_VEL
LIN {X 0,Y 284.599,Z 649.154,A -85,B 0,C 180,E1 -17094.332,E2 -17094.332} C_VEL
LIN {X 0,Y 284.856,Z 649.127,A -85,B 0,C 180,E1 -17098.587,E2 -17098.587} C_VEL
LIN {X 0,Y 284.856,Z 649.118,A -85,B 0,C 180,E1 -17101.414,E2 -17101.414} C_VEL
LIN {X 0,Y 284.688,Z 649.146,A -85,B 0,C 180,E1 -17107.091,E2 -17107.091} C_VEL
LIN {X 0,Y 284.521,Z 649.159,A -85,B 0,C 180,E1 -17109.957,E2 -17109.957} C_VEL
LIN {X 0,Y 284.483,Z 649.166,A -85,B 0,C 180,E1 -17114.303,E2 -17114.303} C_VEL
LIN {X 0,Y 284.425,Z 649.181,A -85,B 0,C 180,E1 -17117.249,E2 -17117.249} C_VEL
LIN {X 0,Y 284.379,Z 649.179,A -85,B 0,C 180,E1 -17120.243,E2 -17120.243} C_VEL
LIN {X 0,Y 284.326,Z 649.184,A -85,B 0,C 180,E1 -17123.855,E2 -17123.855} C_VEL
LIN {X 0,Y 284.29,Z 649.171,A -85,B 0,C 180,E1 -17128.016,E2 -17128.016} C_VEL
LIN {X 0,Y 284.287,Z 649.188,A -85,B 0,C 180,E1 -17131.276,E2 -17131.276} C_VEL
LIN {X 0,Y 284.338,Z 649.193,A -85,B 0,C 180,E1 -17135.347,E2 -17135.347} C_VEL
LIN {X 0,Y 284.3,Z 649.197,A -85,B 0,C 180,E1 -17138.172,E2 -17138.172} C_VEL
LIN {X 0,Y 284.239,Z 649.193,A -85,B 0,C 180,E1 -17142.118,E2 -17142.118} C_VEL
LIN {X 0,Y 284.239,Z 649.195,A -85,B 0,C 180,E1 -17146.186,E2 -17146.186} C_VEL
LIN {X 0,Y 284.272,Z 649.421,A -85,B 0,C 180,E1 -17147.762,E2 -17147.762} C_VEL
LIN {X 0,Y 285.245,Z 652.024,A -85,B 0,C 180,E1 -17148.008,E2 -17148.008} C_VEL
LIN {X 0,Y 287.173,Z 654.647,A -85,B 0,C 180,E1 -17148.407,E2 -17148.407} C_VEL
LIN {X 0,Y 292.407,Z 663.154,A -85,B 0,C 180,E1 -17149.494,E2 -17149.494} C_VEL
LIN {X 0,Y 301.082,Z 679.297,A -85,B 0,C 180,E1 -17151.24,E2 -17151.24} C_VEL
LIN {X 0,Y 308.785,Z 695.892,A -85,B 0,C 180,E1 -17152.74,E2 -17152.74} C_VEL
LIN {X 0,Y 309.179,Z 697.84,A -85,B 0,C 180,E1 -17152.844,E2 -17152.844} C_VEL
LIN {X 0,Y 306.015,Z 784.672,A -85,B 0,C 180,E1 -17154.874,E2 -17154.874} C_VEL
LIN {X 0,Y 304.888,Z 799.312,A -85,B 0,C 180,E1 -17155.465,E2 -17155.465} C_VEL
LIN {X 0,Y 303.437,Z 812.313,A -85,B 0,C 180,E1 -17156.229,E2 -17156.229} C_VEL
LIN {X 0,Y 301.623,Z 824.65,A -85,B 0,C 180,E1 -17157.186,E2 -17157.186} C_VEL
LIN {X 0,Y 299.408,Z 837.758,A -85,B 0,C 180,E1 -17158.515,E2 -17158.515} C_VEL
LIN {X 0,Y 297.069,Z 849.511,A -85,B 0,C 180,E1 -17160.015,E2 -17160.015} C_VEL
LIN {X 0,Y 294.883,Z 859.259,A -85,B 0,C 180,E1 -17161.532,E2 -17161.532} C_VEL
LIN {X 0,Y 292.391,Z 870.023,A -85,B 0,C 180,E1 -17163.598,E2 -17163.598} C_VEL
LIN {X 0,Y 290.071,Z 878.874,A -85,B 0,C 180,E1 -17165.677,E2 -17165.677} C_VEL
LIN {X 0,Y 287.834,Z 887.218,A -85,B 0,C 180,E1 -17168.102,E2 -17168.102} C_VEL
LIN {X 0,Y 286.037,Z 894.101,A -85,B 0,C 180,E1 -17170.628,E2 -17170.628} C_VEL
LIN {X 0,Y 284.792,Z 898.736,A -85,B 0,C 180,E1 -17172.775,E2 -17172.775} C_VEL
LIN {X 0,Y 283.648,Z 903.52,A -85,B 0,C 180,E1 -17175.654,E2 -17175.654} C_VEL
LIN {X 0,Y 282.815,Z 906.801,A -85,B 0,C 180,E1 -17178.533,E2 -17178.533} C_VEL
LIN {X 0,Y 282.539,Z 908.665,A -85,B 0,C 180,E1 -17181.417,E2 -17181.417} C_VEL
LIN {X 0,Y 282.486,Z 909.184,A -85,B 0,C 180,E1 -17184.369,E2 -17184.369} C_VEL
LIN {X 0,Y 282.454,Z 908.419,A -85,B 0,C 180,E1 -17187.148,E2 -17187.148} C_VEL
LIN {X 0,Y 282.537,Z 906.331,A -85,B 0,C 180,E1 -17190,E2 -17190} C_VEL
LIN {X 0,Y 282.939,Z 902.873,A -85,B 0,C 180,E1 -17192.848,E2 -17192.848} C_VEL
LIN {X 0,Y 283.715,Z 899.338,A -85,B 0,C 180,E1 -17194.974,E2 -17194.974} C_VEL
LIN {X 0,Y 284.762,Z 893.165,A -85,B 0,C 180,E1 -17197.802,E2 -17197.802} C_VEL
LIN {X 0,Y 286.093,Z 886.343,A -85,B 0,C 180,E1 -17200.242,E2 -17200.242} C_VEL
LIN {X 0,Y 287.615,Z 877.789,A -85,B 0,C 180,E1 -17202.704,E2 -17202.704} C_VEL
LIN {X 0,Y 289.634,Z 868.871,A -85,B 0,C 180,E1 -17204.761,E2 -17204.761} C_VEL
LIN {X 0,Y 291.753,Z 858.095,A -85,B 0,C 180,E1 -17206.802,E2 -17206.802} C_VEL
LIN {X 0,Y 293.719,Z 847.16,A -85,B 0,C 180,E1 -17208.484,E2 -17208.484} C_VEL
LIN {X 0,Y 295.505,Z 835.168,A -85,B 0,C 180,E1 -17209.992,E2 -17209.992} C_VEL
LIN {X 0,Y 297.184,Z 823.618,A -85,B 0,C 180,E1 -17211.14,E2 -17211.14} C_VEL
LIN {X 0,Y 298.767,Z 809.962,A -85,B 0,C 180,E1 -17212.2,E2 -17212.2} C_VEL
LIN {X 0,Y 299.899,Z 796.414,A -85,B 0,C 180,E1 -17212.975,E2 -17212.975} C_VEL
LIN {X 0,Y 300.715,Z 781.896,A -85,B 0,C 180,E1 -17213.524,E2 -17213.524} C_VEL
LIN {X 0,Y 303.625,Z 692.419,A -85,B 0,C 180,E1 -17215.61,E2 -17215.61} C_VEL
LIN {X 0,Y 301.76,Z 686.988,A -85,B 0,C 180,E1 -17215.95,E2 -17215.95} C_VEL
LIN {X 0,Y 293.914,Z 668.502,A -85,B 0,C 180,E1 -17217.316,E2 -17217.316} C_VEL
LIN {X 0,Y 287.76,Z 656.17,A -85,B 0,C 180,E1 -17218.392,E2 -17218.392} C_VEL
LIN {X 0,Y 285.566,Z 652.478,A -85,B 0,C 180,E1 -17218.77,E2 -17218.77} C_VEL
LIN {X 0,Y 284.38,Z 649.725,A -85,B 0,C 180,E1 -17218.999,E2 -17218.999} C_VEL
LIN {X 0,Y 284.278,Z 649.195,A -85,B 0,C 180,E1 -17219.067,E2 -17219.067} C_VEL
LIN {X 0,Y 284.307,Z 649.196,A -85,B 0,C 180,E1 -17222.945,E2 -17222.945} C_VEL
LIN {X 0,Y 284.321,Z 649.192,A -85,B 0,C 180,E1 -17226.388,E2 -17226.388} C_VEL
LIN {X 0,Y 284.258,Z 649.183,A -85,B 0,C 180,E1 -17230.003,E2 -17230.003} C_VEL
LIN {X 0,Y 284.248,Z 649.197,A -85,B 0,C 180,E1 -17234.19,E2 -17234.19} C_VEL
LIN {X 0,Y 284.242,Z 649.201,A -85,B 0,C 180,E1 -17238.118,E2 -17238.118} C_VEL
LIN {X 0,Y 284.243,Z 649.178,A -85,B 0,C 180,E1 -17241.444,E2 -17241.444} C_VEL
LIN {X 0,Y 283.619,Z 649.253,A -85,B 0,C 180,E1 -17242.626,E2 -17242.626} C_VEL
LIN {X 0,Y 280.772,Z 649.619,A -85,B 0,C 180,E1 -17244.551,E2 -17244.551} C_VEL
LIN {X 0,Y 278.34,Z 649.937,A -85,B 0,C 180,E1 -17246.115,E2 -17246.115} C_VEL
LIN {X 0,Y 277.313,Z 650.067,A -85,B 0,C 180,E1 -17247.327,E2 -17247.327} C_VEL
LIN {X 0,Y 277.24,Z 650.072,A -85,B 0,C 180,E1 -17247.738,E2 -17247.738} C_VEL
LIN {X 0,Y 277.242,Z 650.067,A -85,B 0,C 180,E1 -17251.207,E2 -17251.207} C_VEL
LIN {X 0,Y 277.249,Z 650.068,A -85,B 0,C 180,E1 -17254.473,E2 -17254.473} C_VEL
LIN {X 0,Y 277.263,Z 650.066,A -85,B 0,C 180,E1 -17257.652,E2 -17257.652} C_VEL
LIN {X 0,Y 277.327,Z 650.059,A -85,B 0,C 180,E1 -17260.764,E2 -17260.764} C_VEL
LIN {X 0,Y 277.417,Z 650.051,A -85,B 0,C 180,E1 -17265.324,E2 -17265.324} C_VEL
LIN {X 0,Y 277.46,Z 650.028,A -85,B 0,C 180,E1 -17269.787,E2 -17269.787} C_VEL
LIN {X 0,Y 277.604,Z 650.028,A -85,B 0,C 180,E1 -17272.727,E2 -17272.727} C_VEL
LIN {X 0,Y 277.821,Z 650.002,A -85,B 0,C 180,E1 -17278.55,E2 -17278.55} C_VEL
LIN {X 0,Y 277.822,Z 649.994,A -85,B 0,C 180,E1 -17281.449,E2 -17281.449} C_VEL
LIN {X 0,Y 277.643,Z 650.021,A -85,B 0,C 180,E1 -17287.271,E2 -17287.271} C_VEL
LIN {X 0,Y 277.463,Z 650.039,A -85,B 0,C 180,E1 -17290.213,E2 -17290.213} C_VEL
LIN {X 0,Y 277.437,Z 650.043,A -85,B 0,C 180,E1 -17294.674,E2 -17294.674} C_VEL
LIN {X 0,Y 277.346,Z 650.054,A -85,B 0,C 180,E1 -17299.233,E2 -17299.233} C_VEL
LIN {X 0,Y 277.293,Z 650.061,A -85,B 0,C 180,E1 -17304.157,E2 -17304.157} C_VEL
LIN {X 0,Y 277.327,Z 650.056,A -85,B 0,C 180,E1 -17307.505,E2 -17307.505} C_VEL
LIN {X 0,Y 277.273,Z 650.067,A -85,B 0,C 180,E1 -17310.481,E2 -17310.481} C_VEL
LIN {X 0,Y 277.255,Z 650.07,A -85,B 0,C 180,E1 -17313.894,E2 -17313.894} C_VEL
LIN {X 0,Y 277.289,Z 650.068,A -85,B 0,C 180,E1 -17317.466,E2 -17317.466} C_VEL
LIN {X 0,Y 277.242,Z 650.074,A -85,B 0,C 180,E1 -17321.23,E2 -17321.23} C_VEL
LIN {X 0,Y 277.224,Z 650.076,A -85,B 0,C 180,E1 -17325.221,E2 -17325.221} C_VEL
LIN {X 0,Y 277.223,Z 650.077,A -85,B 0,C 180,E1 -17329.512,E2 -17329.512} C_VEL
LIN {X 0,Y 277.272,Z 650.116,A -85,B 0,C 180,E1 -17330.075,E2 -17330.075} C_VEL
LIN {X 0,Y 279.86,Z 659.89,A -85,B 0,C 180,E1 -17333.475,E2 -17333.475} C_VEL
LIN {X 0,Y 281.367,Z 666.324,A -85,B 0,C 180,E1 -17335.586,E2 -17335.586} C_VEL
LIN {X 0,Y 291.085,Z 688.831,A -85,B 0,C 180,E1 -17337.421,E2 -17337.421} C_VEL
LIN {X 0,Y 292.917,Z 694.026,A -85,B 0,C 180,E1 -17337.773,E2 -17337.773} C_VEL
LIN {X 0,Y 296.641,Z 720.026,A -85,B 0,C 180,E1 -17338.891,E2 -17338.891} C_VEL
LIN {X 0,Y 293.932,Z 803.615,A -85,B 0,C 180,E1 -17340.894,E2 -17340.894} C_VEL
LIN {X 0,Y 292.842,Z 818.183,A -85,B 0,C 180,E1 -17341.462,E2 -17341.462} C_VEL
LIN {X 0,Y 291.291,Z 832.626,A -85,B 0,C 180,E1 -17342.325,E2 -17342.325} C_VEL
LIN {X 0,Y 289.611,Z 845.027,A -85,B 0,C 180,E1 -17343.324,E2 -17343.324} C_VEL
LIN {X 0,Y 287.644,Z 857.524,A -85,B 0,C 180,E1 -17344.619,E2 -17344.619} C_VEL
LIN {X 0,Y 285.461,Z 869.82,A -85,B 0,C 180,E1 -17346.225,E2 -17346.225} C_VEL
LIN {X 0,Y 283.552,Z 879.628,A -85,B 0,C 180,E1 -17347.791,E2 -17347.791} C_VEL
LIN {X 0,Y 281.686,Z 888.836,A -85,B 0,C 180,E1 -17349.555,E2 -17349.555} C_VEL
LIN {X 0,Y 279.78,Z 898.071,A -85,B 0,C 180,E1 -17351.7,E2 -17351.7} C_VEL
LIN {X 0,Y 278.26,Z 905.764,A -85,B 0,C 180,E1 -17353.869,E2 -17353.869} C_VEL
LIN {X 0,Y 277.211,Z 912.186,A -85,B 0,C 180,E1 -17356.063,E2 -17356.063} C_VEL
LIN {X 0,Y 276.24,Z 917.44,A -85,B 0,C 180,E1 -17358.256,E2 -17358.256} C_VEL
LIN {X 0,Y 275.608,Z 922.992,A -85,B 0,C 180,E1 -17361.199,E2 -17361.199} C_VEL
LIN {X 0,Y 275.344,Z 926.939,A -85,B 0,C 180,E1 -17364.14,E2 -17364.14} C_VEL
LIN {X 0,Y 275.318,Z 929.435,A -85,B 0,C 180,E1 -17367.073,E2 -17367.073} C_VEL
LIN {X 0,Y 275.332,Z 930.558,A -85,B 0,C 180,E1 -17370,E2 -17370} C_VEL
LIN {X 0,Y 275.283,Z 930.329,A -85,B 0,C 180,E1 -17372.927,E2 -17372.927} C_VEL
LIN {X 0,Y 275.343,Z 928.76,A -85,B 0,C 180,E1 -17375.86,E2 -17375.86} C_VEL
LIN {X 0,Y 275.634,Z 925.824,A -85,B 0,C 180,E1 -17378.8,E2 -17378.8} C_VEL
LIN {X 0,Y 276.333,Z 921.447,A -85,B 0,C 180,E1 -17381.74,E2 -17381.74} C_VEL
LIN {X 0,Y 277.749,Z 915.517,A -85,B 0,C 180,E1 -17384.657,E2 -17384.657} C_VEL
LIN {X 0,Y 279.233,Z 909.462,A -85,B 0,C 180,E1 -17386.978,E2 -17386.978} C_VEL
LIN {X 0,Y 281.154,Z 901.882,A -85,B 0,C 180,E1 -17389.342,E2 -17389.342} C_VEL
LIN {X 0,Y 283.361,Z 893.544,A -85,B 0,C 180,E1 -17391.459,E2 -17391.459} C_VEL
LIN {X 0,Y 286.013,Z 883.527,A -85,B 0,C 180,E1 -17393.534,E2 -17393.534} C_VEL
LIN {X 0,Y 288.811,Z 872.393,A -85,B 0,C 180,E1 -17395.397,E2 -17395.397} C_VEL
LIN {X 0,Y 291.231,Z 861.121,A -85,B 0,C 180,E1 -17396.934,E2 -17396.934} C_VEL
LIN {X 0,Y 293.552,Z 849.358,A -85,B 0,C 180,E1 -17398.219,E2 -17398.219} C_VEL
LIN {X 0,Y 295.818,Z 836.125,A -85,B 0,C 180,E1 -17399.341,E2 -17399.341} C_VEL
LIN {X 0,Y 297.686,Z 822.413,A -85,B 0,C 180,E1 -17400.209,E2 -17400.209} C_VEL
LIN {X 0,Y 299.108,Z 808.219,A -85,B 0,C 180,E1 -17400.832,E2 -17400.832} C_VEL
LIN {X 0,Y 300.078,Z 788.793,A -85,B 0,C 180,E1 -17401.351,E2 -17401.351} C_VEL
LIN {X 0,Y 302.534,Z 721.06,A -85,B 0,C 180,E1 -17402.945,E2 -17402.945} C_VEL
LIN {X 0,Y 299.298,Z 701.8,A -85,B 0,C 180,E1 -17403.933,E2 -17403.933} C_VEL
LIN {X 0,Y 292.656,Z 687.088,A -85,B 0,C 180,E1 -17405.32,E2 -17405.32} C_VEL
LIN {X 0,Y 286.02,Z 673.907,A -85,B 0,C 180,E1 -17406.75,E2 -17406.75} C_VEL
LIN {X 0,Y 283.425,Z 669.194,A -85,B 0,C 180,E1 -17407.322,E2 -17407.322} C_VEL
LIN {X 0,Y 281.698,Z 665.607,A -85,B 0,C 180,E1 -17407.763,E2 -17407.763} C_VEL
LIN {X 0,Y 279.128,Z 656.349,A -85,B 0,C 180,E1 -17411.277,E2 -17411.277} C_VEL
LIN {X 0,Y 277.258,Z 650.059,A -85,B 0,C 180,E1 -17413.891,E2 -17413.891} C_VEL
LIN {X 0,Y 277.239,Z 650.059,A -85,B 0,C 180,E1 -17417.32,E2 -17417.32} C_VEL
LIN {X 0,Y 277.265,Z 650.071,A -85,B 0,C 180,E1 -17420.678,E2 -17420.678} C_VEL
LIN {X 0,Y 277.304,Z 650.057,A -85,B 0,C 180,E1 -17424.345,E2 -17424.345} C_VEL
LIN {X 0,Y 277.245,Z 650.045,A -85,B 0,C 180,E1 -17427.837,E2 -17427.837} C_VEL
LIN {X 0,Y 277.29,Z 650.065,A -85,B 0,C 180,E1 -17431.213,E2 -17431.213} C_VEL
LIN {X 0,Y 277.318,Z 650.059,A -85,B 0,C 180,E1 -17434.48,E2 -17434.48} C_VEL
LIN {X 0,Y 277.286,Z 650.06,A -85,B 0,C 180,E1 -17437.655,E2 -17437.655} C_VEL
LIN {X 0,Y 277.346,Z 650.057,A -85,B 0,C 180,E1 -17440.767,E2 -17440.767} C_VEL
LIN {X 0,Y 277.435,Z 650.046,A -85,B 0,C 180,E1 -17445.326,E2 -17445.326} C_VEL
LIN {X 0,Y 277.462,Z 650.042,A -85,B 0,C 180,E1 -17449.787,E2 -17449.787} C_VEL
LIN {X 0,Y 277.642,Z 650.026,A -85,B 0,C 180,E1 -17452.729,E2 -17452.729} C_VEL
LIN {X 0,Y 277.822,Z 650.003,A -85,B 0,C 180,E1 -17458.551,E2 -17458.551} C_VEL
LIN {X 0,Y 277.822,Z 649.994,A -85,B 0,C 180,E1 -17461.45,E2 -17461.45} C_VEL
LIN {X 0,Y 277.642,Z 650.025,A -85,B 0,C 180,E1 -17467.272,E2 -17467.272} C_VEL
LIN {X 0,Y 277.463,Z 650.037,A -85,B 0,C 180,E1 -17470.213,E2 -17470.213} C_VEL
LIN {X 0,Y 277.436,Z 650.041,A -85,B 0,C 180,E1 -17474.675,E2 -17474.675} C_VEL
LIN {X 0,Y 277.344,Z 650.052,A -85,B 0,C 180,E1 -17479.234,E2 -17479.234} C_VEL
LIN {X 0,Y 277.288,Z 650.061,A -85,B 0,C 180,E1 -17483.925,E2 -17483.925} C_VEL
LIN {X 0,Y 277.275,Z 650.052,A -85,B 0,C 180,E1 -17487.485,E2 -17487.485} C_VEL
LIN {X 0,Y 277.249,Z 650.051,A -85,B 0,C 180,E1 -17490.473,E2 -17490.473} C_VEL
LIN {X 0,Y 277.247,Z 650.068,A -85,B 0,C 180,E1 -17493.896,E2 -17493.896} C_VEL
LIN {X 0,Y 277.256,Z 650.07,A -85,B 0,C 180,E1 -17497.472,E2 -17497.472} C_VEL
LIN {X 0,Y 277.186,Z 650.063,A -85,B 0,C 180,E1 -17501.242,E2 -17501.242} C_VEL
LIN {X 0,Y 277.196,Z 650.069,A -85,B 0,C 180,E1 -17505.228,E2 -17505.228} C_VEL
LIN {X 0,Y 277.216,Z 650.073,A -85,B 0,C 180,E1 -17506.542,E2 -17506.542} C_VEL
LIN {X 0,Y 278.273,Z 653.04,A -85,B 0,C 180,E1 -17506.849,E2 -17506.849} C_VEL
LIN {X 0,Y 280.045,Z 655.273,A -85,B 0,C 180,E1 -17507.233,E2 -17507.233} C_VEL
LIN {X 0,Y 282.275,Z 658.695,A -85,B 0,C 180,E1 -17507.727,E2 -17507.727} C_VEL
LIN {X 0,Y 289.108,Z 670.006,A -85,B 0,C 180,E1 -17509.195,E2 -17509.195} C_VEL
LIN {X 0,Y 296.773,Z 684.749,A -85,B 0,C 180,E1 -17510.79,E2 -17510.79} C_VEL
LIN {X 0,Y 303.193,Z 698.721,A -85,B 0,C 180,E1 -17512.086,E2 -17512.086} C_VEL
LIN {X 0,Y 300.034,Z 785.075,A -85,B 0,C 180,E1 -17514.155,E2 -17514.155} C_VEL
LIN {X 0,Y 298.948,Z 799.124,A -85,B 0,C 180,E1 -17514.729,E2 -17514.729} C_VEL
LIN {X 0,Y 297.516,Z 811.674,A -85,B 0,C 180,E1 -17515.463,E2 -17515.463} C_VEL
LIN {X 0,Y 295.447,Z 825.222,A -85,B 0,C 180,E1 -17516.526,E2 -17516.526} C_VEL
LIN {X 0,Y 293.292,Z 837.452,A -85,B 0,C 180,E1 -17517.781,E2 -17517.781} C_VEL
LIN {X 0,Y 290.867,Z 849.308,A -85,B 0,C 180,E1 -17519.308,E2 -17519.308} C_VEL
LIN {X 0,Y 288.316,Z 860.186,A -85,B 0,C 180,E1 -17521.036,E2 -17521.036} C_VEL
LIN {X 0,Y 285.95,Z 869.964,A -85,B 0,C 180,E1 -17522.955,E2 -17522.955} C_VEL
LIN {X 0,Y 283.539,Z 878.871,A -85,B 0,C 180,E1 -17525.079,E2 -17525.079} C_VEL
LIN {X 0,Y 281.459,Z 886.259,A -85,B 0,C 180,E1 -17527.231,E2 -17527.231} C_VEL
LIN {X 0,Y 279.793,Z 892.385,A -85,B 0,C 180,E1 -17529.411,E2 -17529.411} C_VEL
LIN {X 0,Y 278.352,Z 897.443,A -85,B 0,C 180,E1 -17531.603,E2 -17531.603} C_VEL
LIN {X 0,Y 277.261,Z 901.473,A -85,B 0,C 180,E1 -17533.81,E2 -17533.81} C_VEL
LIN {X 0,Y 276.213,Z 905.526,A -85,B 0,C 180,E1 -17536.762,E2 -17536.762} C_VEL
LIN {X 0,Y 275.581,Z 908.13,A -85,B 0,C 180,E1 -17539.717,E2 -17539.717} C_VEL
LIN {X 0,Y 275.37,Z 909.361,A -85,B 0,C 180,E1 -17542.669,E2 -17542.669} C_VEL
LIN {X 0,Y 275.409,Z 909.445,A -85,B 0,C 180,E1 -17544.401,E2 -17544.401} C_VEL
LIN {X 0,Y 275.38,Z 908.732,A -85,B 0,C 180,E1 -17547.074,E2 -17547.074} C_VEL
LIN {X 0,Y 275.45,Z 906.677,A -85,B 0,C 180,E1 -17550,E2 -17550} C_VEL
LIN {X 0,Y 275.862,Z 903.253,A -85,B 0,C 180,E1 -17552.921,E2 -17552.921} C_VEL
LIN {X 0,Y 276.648,Z 899.75,A -85,B 0,C 180,E1 -17555.101,E2 -17555.101} C_VEL
LIN {X 0,Y 277.744,Z 893.62,A -85,B 0,C 180,E1 -17558,E2 -17558} C_VEL
LIN {X 0,Y 279.277,Z 886.087,A -85,B 0,C 180,E1 -17560.746,E2 -17560.746} C_VEL
LIN {X 0,Y 280.724,Z 878.335,A -85,B 0,C 180,E1 -17563.022,E2 -17563.022} C_VEL
LIN {X 0,Y 282.807,Z 869.472,A -85,B 0,C 180,E1 -17565.126,E2 -17565.126} C_VEL
LIN {X 0,Y 285.011,Z 858.76,A -85,B 0,C 180,E1 -17567.212,E2 -17567.212} C_VEL
LIN {X 0,Y 287.026,Z 847.907,A -85,B 0,C 180,E1 -17568.931,E2 -17568.931} C_VEL
LIN {X 0,Y 288.886,Z 836.029,A -85,B 0,C 180,E1 -17570.47,E2 -17570.47} C_VEL
LIN {X 0,Y 290.911,Z 822.775,A -85,B 0,C 180,E1 -17571.805,E2 -17571.805} C_VEL
LIN {X 0,Y 292.383,Z 809.997,A -85,B 0,C 180,E1 -17572.805,E2 -17572.805} C_VEL
LIN {X 0,Y 293.569,Z 796.347,A -85,B 0,C 180,E1 -17573.594,E2 -17573.594} C_VEL
LIN {X 0,Y 294.41,Z 781.934,A -85,B 0,C 180,E1 -17574.143,E2 -17574.143} C_VEL
LIN {X 0,Y 297.281,Z 693.34,A -85,B 0,C 180,E1 -17576.258,E2 -17576.258} C_VEL
LIN {X 0,Y 289.118,Z 673.614,A -85,B 0,C 180,E1 -17577.731,E2 -17577.731} C_VEL
LIN {X 0,Y 282.768,Z 660.634,A -85,B 0,C 180,E1 -17578.883,E2 -17578.883} C_VEL
LIN {X 0,Y 277.509,Z 651.271,A -85,B 0,C 180,E1 -17579.846,E2 -17579.846} C_VEL
LIN {X 0,Y 277.258,Z 650.075,A -85,B 0,C 180,E1 -17579.93,E2 -17579.93} C_VEL
LIN {X 0,Y 277.249,Z 650.076,A -85,B 0,C 180,E1 -17583.896,E2 -17583.896} C_VEL
LIN {X 0,Y 277.235,Z 650.077,A -85,B 0,C 180,E1 -17587.475,E2 -17587.475} C_VEL
LIN {X 0,Y 277.191,Z 650.072,A -85,B 0,C 180,E1 -17591.24,E2 -17591.24} C_VEL
LIN {X 0,Y 277.197,Z 650.083,A -85,B 0,C 180,E1 -17595.228,E2 -17595.228} C_VEL
LIN {X 0,Y 277.179,Z 650.083,A -85,B 0,C 180,E1 -17598.757,E2 -17598.757} C_VEL
LIN {X 0,Y 277.236,Z 650.044,A -85,B 0,C 180,E1 -17602.525,E2 -17602.525} C_VEL
LIN {X 0,Y 277.248,Z 650.073,A -85,B 0,C 180,E1 -17606.104,E2 -17606.104} C_VEL
LIN {X 0,Y 277.24,Z 650.072,A -85,B 0,C 180,E1 -17607.738,E2 -17607.738} C_VEL
LIN {X 0,Y 276.601,Z 650.156,A -85,B 0,C 180,E1 -17608.951,E2 -17608.951} C_VEL
LIN {X 0,Y 273.761,Z 650.515,A -85,B 0,C 180,E1 -17610.926,E2 -17610.926} C_VEL
LIN {X 0,Y 271.329,Z 650.815,A -85,B 0,C 180,E1 -17612.531,E2 -17612.531} C_VEL
LIN {X 0,Y 270.277,Z 650.939,A -85,B 0,C 180,E1 -17613.775,E2 -17613.775} C_VEL
LIN {X 0,Y 270.189,Z 650.944,A -85,B 0,C 180,E1 -17614.197,E2 -17614.197} C_VEL
LIN {X 0,Y 270.202,Z 650.939,A -85,B 0,C 180,E1 -17617.035,E2 -17617.035} C_VEL
LIN {X 0,Y 270.263,Z 650.94,A -85,B 0,C 180,E1 -17620.241,E2 -17620.241} C_VEL
LIN {X 0,Y 270.376,Z 650.926,A -85,B 0,C 180,E1 -17624.933,E2 -17624.933} C_VEL
LIN {X 0,Y 270.412,Z 650.906,A -85,B 0,C 180,E1 -17629.517,E2 -17629.517} C_VEL
LIN {X 0,Y 270.565,Z 650.905,A -85,B 0,C 180,E1 -17632.537,E2 -17632.537} C_VEL
LIN {X 0,Y 270.787,Z 650.879,A -85,B 0,C 180,E1 -17638.512,E2 -17638.512} C_VEL
LIN {X 0,Y 270.788,Z 650.87,A -85,B 0,C 180,E1 -17641.487,E2 -17641.487} C_VEL
LIN {X 0,Y 270.601,Z 650.899,A -85,B 0,C 180,E1 -17647.461,E2 -17647.461} C_VEL
LIN {X 0,Y 270.415,Z 650.916,A -85,B 0,C 180,E1 -17650.482,E2 -17650.482} C_VEL
LIN {X 0,Y 270.405,Z 650.918,A -85,B 0,C 180,E1 -17655.064,E2 -17655.064} C_VEL
LIN {X 0,Y 270.303,Z 650.93,A -85,B 0,C 180,E1 -17659.755,E2 -17659.755} C_VEL
LIN {X 0,Y 270.239,Z 650.943,A -85,B 0,C 180,E1 -17664.589,E2 -17664.589} C_VEL
LIN {X 0,Y 270.273,Z 650.936,A -85,B 0,C 180,E1 -17667.908,E2 -17667.908} C_VEL
LIN {X 0,Y 270.186,Z 650.95,A -85,B 0,C 180,E1 -17671.348,E2 -17671.348} C_VEL
LIN {X 0,Y 270.216,Z 650.951,A -85,B 0,C 180,E1 -17674.903,E2 -17674.903} C_VEL
LIN {X 0,Y 270.223,Z 650.948,A -85,B 0,C 180,E1 -17678.717,E2 -17678.717} C_VEL
LIN {X 0,Y 270.2,Z 650.952,A -85,B 0,C 180,E1 -17682.553,E2 -17682.553} C_VEL
LIN {X 0,Y 270.172,Z 650.945,A -85,B 0,C 180,E1 -17686.749,E2 -17686.749} C_VEL
LIN {X 0,Y 270.226,Z 651.158,A -85,B 0,C 180,E1 -17689.359,E2 -17689.359} C_VEL
LIN {X 0,Y 272.921,Z 661.161,A -85,B 0,C 180,E1 -17692.966,E2 -17692.966} C_VEL
LIN {X 0,Y 274.092,Z 666.125,A -85,B 0,C 180,E1 -17694.64,E2 -17694.64} C_VEL
LIN {X 0,Y 283.268,Z 686.782,A -85,B 0,C 180,E1 -17696.437,E2 -17696.437} C_VEL
LIN {X 0,Y 286.912,Z 696.067,A -85,B 0,C 180,E1 -17697.141,E2 -17697.141} C_VEL
LIN {X 0,Y 290.438,Z 721.641,A -85,B 0,C 180,E1 -17698.263,E2 -17698.263} C_VEL
LIN {X 0,Y 287.555,Z 804.504,A -85,B 0,C 180,E1 -17700.285,E2 -17700.285} C_VEL
LIN {X 0,Y 286.432,Z 818.543,A -85,B 0,C 180,E1 -17700.863,E2 -17700.863} C_VEL
LIN {X 0,Y 284.852,Z 832.819,A -85,B 0,C 180,E1 -17701.744,E2 -17701.744} C_VEL
LIN {X 0,Y 282.959,Z 846.008,A -85,B 0,C 180,E1 -17702.845,E2 -17702.845} C_VEL
LIN {X 0,Y 280.918,Z 858.322,A -85,B 0,C 180,E1 -17704.173,E2 -17704.173} C_VEL
LIN {X 0,Y 278.691,Z 870.383,A -85,B 0,C 180,E1 -17705.808,E2 -17705.808} C_VEL
LIN {X 0,Y 276.508,Z 881.036,A -85,B 0,C 180,E1 -17707.588,E2 -17707.588} C_VEL
LIN {X 0,Y 274.289,Z 891.614,A -85,B 0,C 180,E1 -17709.763,E2 -17709.763} C_VEL
LIN {X 0,Y 272.365,Z 900.335,A -85,B 0,C 180,E1 -17711.962,E2 -17711.962} C_VEL
LIN {X 0,Y 271.058,Z 907.595,A -85,B 0,C 180,E1 -17714.202,E2 -17714.202} C_VEL
LIN {X 0,Y 269.905,Z 913.621,A -85,B 0,C 180,E1 -17716.447,E2 -17716.447} C_VEL
LIN {X 0,Y 269.008,Z 918.598,A -85,B 0,C 180,E1 -17718.7,E2 -17718.7} C_VEL
LIN {X 0,Y 268.451,Z 923.738,A -85,B 0,C 180,E1 -17721.721,E2 -17721.721} C_VEL
LIN {X 0,Y 268.234,Z 927.256,A -85,B 0,C 180,E1 -17724.644,E2 -17724.644} C_VEL
LIN {X 0,Y 268.226,Z 929.133,A -85,B 0,C 180,E1 -17726.996,E2 -17726.996} C_VEL
LIN {X 0,Y 268.253,Z 930.28,A -85,B 0,C 180,E1 -17730,E2 -17730} C_VEL
LIN {X 0,Y 268.194,Z 930.073,A -85,B 0,C 180,E1 -17733.004,E2 -17733.004} C_VEL
LIN {X 0,Y 268.244,Z 928.526,A -85,B 0,C 180,E1 -17736.016,E2 -17736.016} C_VEL
LIN {X 0,Y 268.597,Z 925.615,A -85,B 0,C 180,E1 -17739.032,E2 -17739.032} C_VEL
LIN {X 0,Y 269.335,Z 921.262,A -85,B 0,C 180,E1 -17742.049,E2 -17742.049} C_VEL
LIN {X 0,Y 270.833,Z 915.359,A -85,B 0,C 180,E1 -17745.04,E2 -17745.04} C_VEL
LIN {X 0,Y 272.449,Z 909.179,A -85,B 0,C 180,E1 -17747.473,E2 -17747.473} C_VEL
LIN {X 0,Y 274.435,Z 901.788,A -85,B 0,C 180,E1 -17749.835,E2 -17749.835} C_VEL
LIN {X 0,Y 276.738,Z 893.489,A -85,B 0,C 180,E1 -17751.999,E2 -17751.999} C_VEL
LIN {X 0,Y 279.519,Z 883.517,A -85,B 0,C 180,E1 -17754.115,E2 -17754.115} C_VEL
LIN {X 0,Y 282.408,Z 872.446,A -85,B 0,C 180,E1 -17756.015,E2 -17756.015} C_VEL
LIN {X 0,Y 284.872,Z 861.443,A -85,B 0,C 180,E1 -17757.556,E2 -17757.556} C_VEL
LIN {X 0,Y 287.324,Z 849.572,A -85,B 0,C 180,E1 -17758.887,E2 -17758.887} C_VEL
LIN {X 0,Y 289.682,Z 836.518,A -85,B 0,C 180,E1 -17760.025,E2 -17760.025} C_VEL
LIN {X 0,Y 291.606,Z 823.043,A -85,B 0,C 180,E1 -17760.907,E2 -17760.907} C_VEL
LIN {X 0,Y 293.072,Z 809.296,A -85,B 0,C 180,E1 -17761.539,E2 -17761.539} C_VEL
LIN {X 0,Y 293.966,Z 793.229,A -85,B 0,C 180,E1 -17762.006,E2 -17762.006} C_VEL
LIN {X 0,Y 296.646,Z 721.728,A -85,B 0,C 180,E1 -17763.72,E2 -17763.72} C_VEL
LIN {X 0,Y 293.769,Z 704.589,A -85,B 0,C 180,E1 -17764.631,E2 -17764.631} C_VEL
LIN {X 0,Y 287.465,Z 690.605,A -85,B 0,C 180,E1 -17766,E2 -17766} C_VEL
LIN {X 0,Y 281.194,Z 677.96,A -85,B 0,C 180,E1 -17767.409,E2 -17767.409} C_VEL
LIN {X 0,Y 276.067,Z 668.729,A -85,B 0,C 180,E1 -17768.595,E2 -17768.595} C_VEL
LIN {X 0,Y 274.386,Z 665.295,A -85,B 0,C 180,E1 -17769.033,E2 -17769.033} C_VEL
LIN {X 0,Y 271.794,Z 656.286,A -85,B 0,C 180,E1 -17772.649,E2 -17772.649} C_VEL
LIN {X 0,Y 270.206,Z 650.943,A -85,B 0,C 180,E1 -17774.966,E2 -17774.966} C_VEL
LIN {X 0,Y 270.213,Z 650.945,A -85,B 0,C 180,E1 -17779.441,E2 -17779.441} C_VEL
LIN {X 0,Y 270.256,Z 650.926,A -85,B 0,C 180,E1 -17783.722,E2 -17783.722} C_VEL
LIN {X 0,Y 270.204,Z 650.934,A -85,B 0,C 180,E1 -17786.893,E2 -17786.893} C_VEL
LIN {X 0,Y 270.229,Z 650.931,A -85,B 0,C 180,E1 -17790.387,E2 -17790.387} C_VEL
LIN {X 0,Y 270.266,Z 650.934,A -85,B 0,C 180,E1 -17793.764,E2 -17793.764} C_VEL
LIN {X 0,Y 270.237,Z 650.939,A -85,B 0,C 180,E1 -17797.039,E2 -17797.039} C_VEL
LIN {X 0,Y 270.302,Z 650.937,A -85,B 0,C 180,E1 -17800.245,E2 -17800.245} C_VEL
LIN {X 0,Y 270.404,Z 650.924,A -85,B 0,C 180,E1 -17804.936,E2 -17804.936} C_VEL
LIN {X 0,Y 270.414,Z 650.923,A -85,B 0,C 180,E1 -17809.518,E2 -17809.518} C_VEL
LIN {X 0,Y 270.6,Z 650.901,A -85,B 0,C 180,E1 -17812.539,E2 -17812.539} C_VEL
LIN {X 0,Y 270.788,Z 650.879,A -85,B 0,C 180,E1 -17818.513,E2 -17818.513} C_VEL
LIN {X 0,Y 270.788,Z 650.87,A -85,B 0,C 180,E1 -17821.488,E2 -17821.488} C_VEL
LIN {X 0,Y 270.6,Z 650.902,A -85,B 0,C 180,E1 -17827.462,E2 -17827.462} C_VEL
LIN {X 0,Y 270.414,Z 650.914,A -85,B 0,C 180,E1 -17830.483,E2 -17830.483} C_VEL
LIN {X 0,Y 270.405,Z 650.916,A -85,B 0,C 180,E1 -17835.065,E2 -17835.065} C_VEL
LIN {X 0,Y 270.302,Z 650.93,A -85,B 0,C 180,E1 -17839.756,E2 -17839.756} C_VEL
LIN {X 0,Y 270.23,Z 650.944,A -85,B 0,C 180,E1 -17844.59,E2 -17844.59} C_VEL
LIN {X 0,Y 270.204,Z 650.925,A -85,B 0,C 180,E1 -17847.917,E2 -17847.917} C_VEL
LIN {X 0,Y 270.175,Z 650.946,A -85,B 0,C 180,E1 -17851.35,E2 -17851.35} C_VEL
LIN {X 0,Y 270.2,Z 650.95,A -85,B 0,C 180,E1 -17854.906,E2 -17854.906} C_VEL
LIN {X 0,Y 270.199,Z 650.953,A -85,B 0,C 180,E1 -17858.711,E2 -17858.711} C_VEL
LIN {X 0,Y 270.159,Z 650.962,A -85,B 0,C 180,E1 -17863.248,E2 -17863.248} C_VEL
LIN {X 0,Y 270.176,Z 650.943,A -85,B 0,C 180,E1 -17865.254,E2 -17865.254} C_VEL
LIN {X 0,Y 271.164,Z 653.826,A -85,B 0,C 180,E1 -17865.574,E2 -17865.574} C_VEL
LIN {X 0,Y 273.084,Z 656.206,A -85,B 0,C 180,E1 -17866.017,E2 -17866.017} C_VEL
LIN {X 0,Y 275.318,Z 659.614,A -85,B 0,C 180,E1 -17866.542,E2 -17866.542} C_VEL
LIN {X 0,Y 282.758,Z 671.358,A -85,B 0,C 180,E1 -17868.216,E2 -17868.216} C_VEL
LIN {X 0,Y 291.186,Z 687.401,A -85,B 0,C 180,E1 -17870.048,E2 -17870.048} C_VEL
LIN {X 0,Y 297.395,Z 701.092,A -85,B 0,C 180,E1 -17871.36,E2 -17871.36} C_VEL
LIN {X 0,Y 294.092,Z 785.822,A -85,B 0,C 180,E1 -17873.421,E2 -17873.421} C_VEL
LIN {X 0,Y 292.857,Z 800.468,A -85,B 0,C 180,E1 -17874.041,E2 -17874.041} C_VEL
LIN {X 0,Y 291.195,Z 814.086,A -85,B 0,C 180,E1 -17874.887,E2 -17874.887} C_VEL
LIN {X 0,Y 289.3,Z 825.903,A -85,B 0,C 180,E1 -17875.85,E2 -17875.85} C_VEL
LIN {X 0,Y 286.949,Z 838.586,A -85,B 0,C 180,E1 -17877.188,E2 -17877.188} C_VEL
LIN {X 0,Y 284.439,Z 850.288,A -85,B 0,C 180,E1 -17878.743,E2 -17878.743} C_VEL
LIN {X 0,Y 281.852,Z 860.819,A -85,B 0,C 180,E1 -17880.464,E2 -17880.464} C_VEL
LIN {X 0,Y 279.123,Z 871.543,A -85,B 0,C 180,E1 -17882.644,E2 -17882.644} C_VEL
LIN {X 0,Y 276.629,Z 880.229,A -85,B 0,C 180,E1 -17884.815,E2 -17884.815} C_VEL
LIN {X 0,Y 274.176,Z 888.526,A -85,B 0,C 180,E1 -17887.388,E2 -17887.388} C_VEL
LIN {X 0,Y 272.494,Z 894.283,A -85,B 0,C 180,E1 -17889.624,E2 -17889.624} C_VEL
LIN {X 0,Y 271.067,Z 898.996,A -85,B 0,C 180,E1 -17891.873,E2 -17891.873} C_VEL
LIN {X 0,Y 269.751,Z 903.854,A -85,B 0,C 180,E1 -17894.898,E2 -17894.898} C_VEL
LIN {X 0,Y 268.774,Z 907.206,A -85,B 0,C 180,E1 -17897.925,E2 -17897.925} C_VEL
LIN {X 0,Y 268.4,Z 909.154,A -85,B 0,C 180,E1 -17900.961,E2 -17900.961} C_VEL
LIN {X 0,Y 268.297,Z 909.757,A -85,B 0,C 180,E1 -17903.986,E2 -17903.986} C_VEL
LIN {X 0,Y 268.285,Z 909.046,A -85,B 0,C 180,E1 -17906.997,E2 -17906.997} C_VEL
LIN {X 0,Y 268.365,Z 907.023,A -85,B 0,C 180,E1 -17910,E2 -17910} C_VEL
LIN {X 0,Y 268.787,Z 903.633,A -85,B 0,C 180,E1 -17912.998,E2 -17912.998} C_VEL
LIN {X 0,Y 269.582,Z 900.157,A -85,B 0,C 180,E1 -17915.235,E2 -17915.235} C_VEL
LIN {X 0,Y 270.426,Z 895.738,A -85,B 0,C 180,E1 -17917.466,E2 -17917.466} C_VEL
LIN {X 0,Y 271.55,Z 890.367,A -85,B 0,C 180,E1 -17919.685,E2 -17919.685} C_VEL
LIN {X 0,Y 273.084,Z 882.697,A -85,B 0,C 180,E1 -17922.258,E2 -17922.258} C_VEL
LIN {X 0,Y 274.922,Z 874.677,A -85,B 0,C 180,E1 -17924.433,E2 -17924.433} C_VEL
LIN {X 0,Y 277.133,Z 865.007,A -85,B 0,C 180,E1 -17926.577,E2 -17926.577} C_VEL
LIN {X 0,Y 279.27,Z 854.291,A -85,B 0,C 180,E1 -17928.525,E2 -17928.525} C_VEL
LIN {X 0,Y 281.434,Z 842.413,A -85,B 0,C 180,E1 -17930.273,E2 -17930.273} C_VEL
LIN {X 0,Y 283.307,Z 830.721,A -85,B 0,C 180,E1 -17931.654,E2 -17931.654} C_VEL
LIN {X 0,Y 285.194,Z 817.923,A -85,B 0,C 180,E1 -17932.838,E2 -17932.838} C_VEL
LIN {X 0,Y 286.566,Z 804.845,A -85,B 0,C 180,E1 -17933.774,E2 -17933.774} C_VEL
LIN {X 0,Y 287.659,Z 790.635,A -85,B 0,C 180,E1 -17934.493,E2 -17934.493} C_VEL
LIN {X 0,Y 288.365,Z 774.674,A -85,B 0,C 180,E1 -17934.984,E2 -17934.984} C_VEL
LIN {X 0,Y 291.105,Z 695.177,A -85,B 0,C 180,E1 -17936.894,E2 -17936.894} C_VEL
LIN {X 0,Y 282.912,Z 675.53,A -85,B 0,C 180,E1 -17938.429,E2 -17938.429} C_VEL
LIN {X 0,Y 277.417,Z 664.433,A -85,B 0,C 180,E1 -17939.461,E2 -17939.461} C_VEL
LIN {X 0,Y 271.594,Z 654.389,A -85,B 0,C 180,E1 -17940.56,E2 -17940.56} C_VEL
LIN {X 0,Y 270.296,Z 651.656,A -85,B 0,C 180,E1 -17940.829,E2 -17940.829} C_VEL
LIN {X 0,Y 270.179,Z 650.957,A -85,B 0,C 180,E1 -17940.908,E2 -17940.908} C_VEL
LIN {X 0,Y 270.2,Z 650.953,A -85,B 0,C 180,E1 -17944.906,E2 -17944.906} C_VEL
LIN {X 0,Y 270.17,Z 650.944,A -85,B 0,C 180,E1 -17948.702,E2 -17948.702} C_VEL
LIN {X 0,Y 270.165,Z 650.954,A -85,B 0,C 180,E1 -17953.248,E2 -17953.248} C_VEL
LIN {X 0,Y 270.153,Z 650.954,A -85,B 0,C 180,E1 -17957.437,E2 -17957.437} C_VEL
LIN {X 0,Y 270.156,Z 650.935,A -85,B 0,C 180,E1 -17961.365,E2 -17961.365} C_VEL
LIN {X 0,Y 270.2,Z 650.94,A -85,B 0,C 180,E1 -17965.094,E2 -17965.094} C_VEL
LIN {X 0,Y 270.187,Z 650.942,A -85,B 0,C 180,E1 -17969.136,E2 -17969.136} C_VEL
LIN {X 0,Y 270.225,Z 650.948,A -85,B 0,C 180,E1 -17972.162,E2 -17972.162} C_VEL
LIN {X 0,Y 270.189,Z 650.944,A -85,B 0,C 180,E1 -17974.197,E2 -17974.197} C_VEL
LIN {X 0,Y 269.515,Z 651.023,A -85,B 0,C 180,E1 -17975.441,E2 -17975.441} C_VEL
LIN {X 0,Y 266.68,Z 651.382,A -85,B 0,C 180,E1 -17977.47,E2 -17977.47} C_VEL
LIN {X 0,Y 264.29,Z 651.689,A -85,B 0,C 180,E1 -17979.119,E2 -17979.119} C_VEL
LIN {X 0,Y 263.28,Z 651.81,A -85,B 0,C 180,E1 -17980.396,E2 -17980.396} C_VEL
LIN {X 0,Y 263.206,Z 651.81,A -85,B 0,C 180,E1 -17980.829,E2 -17980.829} C_VEL
LIN {X 0,Y 263.317,Z 651.805,A -85,B 0,C 180,E1 -17984.519,E2 -17984.519} C_VEL
LIN {X 0,Y 263.352,Z 651.785,A -85,B 0,C 180,E1 -17989.233,E2 -17989.233} C_VEL
LIN {X 0,Y 263.529,Z 651.782,A -85,B 0,C 180,E1 -17992.337,E2 -17992.337} C_VEL
LIN {X 0,Y 263.751,Z 651.755,A -85,B 0,C 180,E1 -17998.473,E2 -17998.473} C_VEL
LIN {X 0,Y 263.752,Z 651.746,A -85,B 0,C 180,E1 -18001.526,E2 -18001.526} C_VEL
LIN {X 0,Y 263.56,Z 651.778,A -85,B 0,C 180,E1 -18007.662,E2 -18007.662} C_VEL
LIN {X 0,Y 263.357,Z 651.794,A -85,B 0,C 180,E1 -18010.766,E2 -18010.766} C_VEL
LIN {X 0,Y 263.353,Z 651.795,A -85,B 0,C 180,E1 -18015.477,E2 -18015.477} C_VEL
LIN {X 0,Y 263.264,Z 651.809,A -85,B 0,C 180,E1 -18020.306,E2 -18020.306} C_VEL
LIN {X 0,Y 263.194,Z 651.822,A -85,B 0,C 180,E1 -18025.292,E2 -18025.292} C_VEL
LIN {X 0,Y 263.181,Z 651.827,A -85,B 0,C 180,E1 -18028.729,E2 -18028.729} C_VEL
LIN {X 0,Y 263.135,Z 651.833,A -85,B 0,C 180,E1 -18032.288,E2 -18032.288} C_VEL
LIN {X 0,Y 263.19,Z 651.827,A -85,B 0,C 180,E1 -18035.977,E2 -18035.977} C_VEL
LIN {X 0,Y 263.155,Z 651.827,A -85,B 0,C 180,E1 -18039.863,E2 -18039.863} C_VEL
LIN {X 0,Y 263.138,Z 651.829,A -85,B 0,C 180,E1 -18043.981,E2 -18043.981} C_VEL
LIN {X 0,Y 263.126,Z 651.834,A -85,B 0,C 180,E1 -18048.406,E2 -18048.406} C_VEL
LIN {X 0,Y 265.644,Z 660.973,A -85,B 0,C 180,E1 -18051.913,E2 -18051.913} C_VEL
LIN {X 0,Y 266.811,Z 665.822,A -85,B 0,C 180,E1 -18053.613,E2 -18053.613} C_VEL
LIN {X 0,Y 274.323,Z 682.197,A -85,B 0,C 180,E1 -18055.162,E2 -18055.162} C_VEL
LIN {X 0,Y 280.957,Z 698.194,A -85,B 0,C 180,E1 -18056.486,E2 -18056.486} C_VEL
LIN {X 0,Y 284.229,Z 721.71,A -85,B 0,C 180,E1 -18057.559,E2 -18057.559} C_VEL
LIN {X 0,Y 281.297,Z 803.977,A -85,B 0,C 180,E1 -18059.607,E2 -18059.607} C_VEL
LIN {X 0,Y 280.136,Z 818.121,A -85,B 0,C 180,E1 -18060.195,E2 -18060.195} C_VEL
LIN {X 0,Y 278.61,Z 831.872,A -85,B 0,C 180,E1 -18061.052,E2 -18061.052} C_VEL
LIN {X 0,Y 276.619,Z 845.204,A -85,B 0,C 180,E1 -18062.17,E2 -18062.17} C_VEL
LIN {X 0,Y 274.358,Z 858.39,A -85,B 0,C 180,E1 -18063.618,E2 -18063.618} C_VEL
LIN {X 0,Y 272.121,Z 869.751,A -85,B 0,C 180,E1 -18065.185,E2 -18065.185} C_VEL
LIN {X 0,Y 269.916,Z 880.469,A -85,B 0,C 180,E1 -18067.01,E2 -18067.01} C_VEL
LIN {X 0,Y 267.931,Z 889.449,A -85,B 0,C 180,E1 -18068.858,E2 -18068.858} C_VEL
LIN {X 0,Y 265.9,Z 898.49,A -85,B 0,C 180,E1 -18071.108,E2 -18071.108} C_VEL
LIN {X 0,Y 264.225,Z 906.112,A -85,B 0,C 180,E1 -18073.42,E2 -18073.42} C_VEL
LIN {X 0,Y 263.277,Z 911.343,A -85,B 0,C 180,E1 -18075.309,E2 -18075.309} C_VEL
LIN {X 0,Y 262.248,Z 916.654,A -85,B 0,C 180,E1 -18077.62,E2 -18077.62} C_VEL
LIN {X 0,Y 261.484,Z 922.262,A -85,B 0,C 180,E1 -18080.72,E2 -18080.72} C_VEL
LIN {X 0,Y 261.16,Z 926.281,A -85,B 0,C 180,E1 -18083.82,E2 -18083.82} C_VEL
LIN {X 0,Y 261.137,Z 928.831,A -85,B 0,C 180,E1 -18086.914,E2 -18086.914} C_VEL
LIN {X 0,Y 261.176,Z 930.001,A -85,B 0,C 180,E1 -18090,E2 -18090} C_VEL
LIN {X 0,Y 261.107,Z 929.817,A -85,B 0,C 180,E1 -18093.086,E2 -18093.086} C_VEL
LIN {X 0,Y 261.156,Z 928.292,A -85,B 0,C 180,E1 -18096.179,E2 -18096.179} C_VEL
LIN {X 0,Y 261.537,Z 925.404,A -85,B 0,C 180,E1 -18099.278,E2 -18099.278} C_VEL
LIN {X 0,Y 262.346,Z 921.079,A -85,B 0,C 180,E1 -18102.375,E2 -18102.375} C_VEL
LIN {X 0,Y 263.941,Z 915.203,A -85,B 0,C 180,E1 -18105.442,E2 -18105.442} C_VEL
LIN {X 0,Y 265.565,Z 909.321,A -85,B 0,C 180,E1 -18107.837,E2 -18107.837} C_VEL
LIN {X 0,Y 267.723,Z 901.696,A -85,B 0,C 180,E1 -18110.354,E2 -18110.354} C_VEL
LIN {X 0,Y 270.114,Z 893.435,A -85,B 0,C 180,E1 -18112.568,E2 -18112.568} C_VEL
LIN {X 0,Y 273.054,Z 883.507,A -85,B 0,C 180,E1 -18114.724,E2 -18114.724} C_VEL
LIN {X 0,Y 276.034,Z 872.491,A -85,B 0,C 180,E1 -18116.663,E2 -18116.663} C_VEL
LIN {X 0,Y 278.524,Z 861.826,A -85,B 0,C 180,E1 -18118.196,E2 -18118.196} C_VEL
LIN {X 0,Y 281.146,Z 849.769,A -85,B 0,C 180,E1 -18119.584,E2 -18119.584} C_VEL
LIN {X 0,Y 283.583,Z 836.87,A -85,B 0,C 180,E1 -18120.74,E2 -18120.74} C_VEL
LIN {X 0,Y 285.561,Z 823.655,A -85,B 0,C 180,E1 -18121.636,E2 -18121.636} C_VEL
LIN {X 0,Y 287.176,Z 809.239,A -85,B 0,C 180,E1 -18122.315,E2 -18122.315} C_VEL
LIN {X 0,Y 288.083,Z 793.595,A -85,B 0,C 180,E1 -18122.783,E2 -18122.783} C_VEL
LIN {X 0,Y 290.866,Z 722.794,A -85,B 0,C 180,E1 -18124.506,E2 -18124.506} C_VEL
LIN {X 0,Y 288.378,Z 707.634,A -85,B 0,C 180,E1 -18125.335,E2 -18125.335} C_VEL
LIN {X 0,Y 281.796,Z 692.934,A -85,B 0,C 180,E1 -18126.828,E2 -18126.828} C_VEL
LIN {X 0,Y 275.009,Z 679.281,A -85,B 0,C 180,E1 -18128.428,E2 -18128.428} C_VEL
LIN {X 0,Y 269.26,Z 669.081,A -85,B 0,C 180,E1 -18129.833,E2 -18129.833} C_VEL
LIN {X 0,Y 267.021,Z 664.849,A -85,B 0,C 180,E1 -18130.46,E2 -18130.46} C_VEL
LIN {X 0,Y 264.449,Z 656.185,A -85,B 0,C 180,E1 -18134.148,E2 -18134.148} C_VEL
LIN {X 0,Y 263.135,Z 651.828,A -85,B 0,C 180,E1 -18136.148,E2 -18136.148} C_VEL
LIN {X 0,Y 263.14,Z 651.833,A -85,B 0,C 180,E1 -18140.134,E2 -18140.134} C_VEL
LIN {X 0,Y 263.188,Z 651.81,A -85,B 0,C 180,E1 -18144.022,E2 -18144.022} C_VEL
LIN {X 0,Y 263.133,Z 651.803,A -85,B 0,C 180,E1 -18147.712,E2 -18147.712} C_VEL
LIN {X 0,Y 263.202,Z 651.823,A -85,B 0,C 180,E1 -18151.783,E2 -18151.783} C_VEL
LIN {X 0,Y 263.232,Z 651.817,A -85,B 0,C 180,E1 -18155.198,E2 -18155.198} C_VEL
LIN {X 0,Y 263.264,Z 651.817,A -85,B 0,C 180,E1 -18159.694,E2 -18159.694} C_VEL
LIN {X 0,Y 263.352,Z 651.804,A -85,B 0,C 180,E1 -18164.522,E2 -18164.522} C_VEL
LIN {X 0,Y 263.356,Z 651.804,A -85,B 0,C 180,E1 -18169.234,E2 -18169.234} C_VEL
LIN {X 0,Y 263.559,Z 651.775,A -85,B 0,C 180,E1 -18172.338,E2 -18172.338} C_VEL
LIN {X 0,Y 263.752,Z 651.756,A -85,B 0,C 180,E1 -18178.474,E2 -18178.474} C_VEL
LIN {X 0,Y 263.752,Z 651.747,A -85,B 0,C 180,E1 -18181.527,E2 -18181.527} C_VEL
LIN {X 0,Y 263.56,Z 651.779,A -85,B 0,C 180,E1 -18187.662,E2 -18187.662} C_VEL
LIN {X 0,Y 263.357,Z 651.794,A -85,B 0,C 180,E1 -18190.767,E2 -18190.767} C_VEL
LIN {X 0,Y 263.352,Z 651.795,A -85,B 0,C 180,E1 -18195.478,E2 -18195.478} C_VEL
LIN {X 0,Y 263.264,Z 651.809,A -85,B 0,C 180,E1 -18200.307,E2 -18200.307} C_VEL
LIN {X 0,Y 263.176,Z 651.829,A -85,B 0,C 180,E1 -18205.295,E2 -18205.295} C_VEL
LIN {X 0,Y 263.137,Z 651.798,A -85,B 0,C 180,E1 -18208.735,E2 -18208.735} C_VEL
LIN {X 0,Y 263.13,Z 651.834,A -85,B 0,C 180,E1 -18212.289,E2 -18212.289} C_VEL
LIN {X 0,Y 263.177,Z 651.823,A -85,B 0,C 180,E1 -18216.762,E2 -18216.762} C_VEL
LIN {X 0,Y 263.092,Z 651.822,A -85,B 0,C 180,E1 -18219.876,E2 -18219.876} C_VEL
LIN {X 0,Y 263.122,Z 651.951,A -85,B 0,C 180,E1 -18223.91,E2 -18223.91} C_VEL
LIN {X 0,Y 264.027,Z 654.568,A -85,B 0,C 180,E1 -18224.193,E2 -18224.193} C_VEL
LIN {X 0,Y 266.201,Z 657.246,A -85,B 0,C 180,E1 -18224.73,E2 -18224.73} C_VEL
LIN {X 0,Y 268.408,Z 660.587,A -85,B 0,C 180,E1 -18225.283,E2 -18225.283} C_VEL
LIN {X 0,Y 276.679,Z 673.337,A -85,B 0,C 180,E1 -18227.245,E2 -18227.245} C_VEL
LIN {X 0,Y 284.077,Z 686.954,A -85,B 0,C 180,E1 -18228.929,E2 -18228.929} C_VEL
LIN {X 0,Y 290.369,Z 700.385,A -85,B 0,C 180,E1 -18230.321,E2 -18230.321} C_VEL
LIN {X 0,Y 291.601,Z 703.234,A -85,B 0,C 180,E1 -18230.59,E2 -18230.59} C_VEL
LIN {X 0,Y 288.289,Z 785.362,A -85,B 0,C 180,E1 -18232.615,E2 -18232.615} C_VEL
LIN {X 0,Y 287.118,Z 799.516,A -85,B 0,C 180,E1 -18233.206,E2 -18233.206} C_VEL
LIN {X 0,Y 285.338,Z 813.716,A -85,B 0,C 180,E1 -18234.081,E2 -18234.081} C_VEL
LIN {X 0,Y 283.387,Z 825.232,A -85,B 0,C 180,E1 -18235.007,E2 -18235.007} C_VEL
LIN {X 0,Y 280.948,Z 838.284,A -85,B 0,C 180,E1 -18236.395,E2 -18236.395} C_VEL
LIN {X 0,Y 278.311,Z 850.088,A -85,B 0,C 180,E1 -18237.974,E2 -18237.974} C_VEL
LIN {X 0,Y 275.542,Z 860.917,A -85,B 0,C 180,E1 -18239.765,E2 -18239.765} C_VEL
LIN {X 0,Y 272.748,Z 871.49,A -85,B 0,C 180,E1 -18241.949,E2 -18241.949} C_VEL
LIN {X 0,Y 270.13,Z 880.231,A -85,B 0,C 180,E1 -18244.165,E2 -18244.165} C_VEL
LIN {X 0,Y 267.531,Z 888.587,A -85,B 0,C 180,E1 -18246.794,E2 -18246.794} C_VEL
LIN {X 0,Y 265.747,Z 894.376,A -85,B 0,C 180,E1 -18249.083,E2 -18249.083} C_VEL
LIN {X 0,Y 264.242,Z 899.129,A -85,B 0,C 180,E1 -18251.388,E2 -18251.388} C_VEL
LIN {X 0,Y 262.819,Z 904.022,A -85,B 0,C 180,E1 -18254.49,E2 -18254.49} C_VEL
LIN {X 0,Y 261.777,Z 907.408,A -85,B 0,C 180,E1 -18257.598,E2 -18257.598} C_VEL
LIN {X 0,Y 261.339,Z 909.391,A -85,B 0,C 180,E1 -18260.715,E2 -18260.715} C_VEL
LIN {X 0,Y 261.217,Z 910.033,A -85,B 0,C 180,E1 -18263.822,E2 -18263.822} C_VEL
LIN {X 0,Y 261.193,Z 909.359,A -85,B 0,C 180,E1 -18266.915,E2 -18266.915} C_VEL
LIN {X 0,Y 261.283,Z 907.368,A -85,B 0,C 180,E1 -18270,E2 -18270} C_VEL
LIN {X 0,Y 261.714,Z 904.013,A -85,B 0,C 180,E1 -18273.079,E2 -18273.079} C_VEL
LIN {X 0,Y 262.519,Z 900.556,A -85,B 0,C 180,E1 -18275.377,E2 -18275.377} C_VEL
LIN {X 0,Y 263.408,Z 896.172,A -85,B 0,C 180,E1 -18277.667,E2 -18277.667} C_VEL
LIN {X 0,Y 264.593,Z 890.839,A -85,B 0,C 180,E1 -18279.942,E2 -18279.942} C_VEL
LIN {X 0,Y 266.17,Z 883.215,A -85,B 0,C 180,E1 -18282.582,E2 -18282.582} C_VEL
LIN {X 0,Y 268.098,Z 875.243,A -85,B 0,C 180,E1 -18284.809,E2 -18284.809} C_VEL
LIN {X 0,Y 270.362,Z 865.634,A -85,B 0,C 180,E1 -18287.004,E2 -18287.004} C_VEL
LIN {X 0,Y 272.604,Z 854.986,A -85,B 0,C 180,E1 -18288.995,E2 -18288.995} C_VEL
LIN {X 0,Y 274.828,Z 843.198,A -85,B 0,C 180,E1 -18290.782,E2 -18290.782} C_VEL
LIN {X 0,Y 276.768,Z 831.62,A -85,B 0,C 180,E1 -18292.193,E2 -18292.193} C_VEL
LIN {X 0,Y 278.857,Z 817.995,A -85,B 0,C 180,E1 -18293.486,E2 -18293.486} C_VEL
LIN {X 0,Y 280.318,Z 804.105,A -85,B 0,C 180,E1 -18294.486,E2 -18294.486} C_VEL
LIN {X 0,Y 281.454,Z 789.559,A -85,B 0,C 180,E1 -18295.208,E2 -18295.208} C_VEL
LIN {X 0,Y 282.263,Z 770.987,A -85,B 0,C 180,E1 -18295.753,E2 -18295.753} C_VEL
LIN {X 0,Y 284.865,Z 696.959,A -85,B 0,C 180,E1 -18297.57,E2 -18297.57} C_VEL
LIN {X 0,Y 277.579,Z 679.317,A -85,B 0,C 180,E1 -18298.993,E2 -18298.993} C_VEL
LIN {X 0,Y 272.429,Z 668.778,A -85,B 0,C 180,E1 -18299.999,E2 -18299.999} C_VEL
LIN {X 0,Y 266.309,Z 658.246,A -85,B 0,C 180,E1 -18301.196,E2 -18301.196} C_VEL
LIN {X 0,Y 264.802,Z 655.61,A -85,B 0,C 180,E1 -18301.504,E2 -18301.504} C_VEL
LIN {X 0,Y 263.38,Z 653.061,A -85,B 0,C 180,E1 -18301.8,E2 -18301.8} C_VEL
LIN {X 0,Y 263.136,Z 651.835,A -85,B 0,C 180,E1 -18301.928,E2 -18301.928} C_VEL
LIN {X 0,Y 263.157,Z 651.829,A -85,B 0,C 180,E1 -18305.983,E2 -18305.983} C_VEL
LIN {X 0,Y 263.078,Z 651.82,A -85,B 0,C 180,E1 -18309.878,E2 -18309.878} C_VEL
LIN {X 0,Y 263.105,Z 651.83,A -85,B 0,C 180,E1 -18313.988,E2 -18313.988} C_VEL
LIN {X 0,Y 263.078,Z 651.838,A -85,B 0,C 180,E1 -18318.097,E2 -18318.097} C_VEL
LIN {X 0,Y 263.107,Z 651.804,A -85,B 0,C 180,E1 -18322.093,E2 -18322.093} C_VEL
LIN {X 0,Y 263.154,Z 651.828,A -85,B 0,C 180,E1 -18325.885,E2 -18325.885} C_VEL
LIN {X 0,Y 263.128,Z 651.819,A -85,B 0,C 180,E1 -18329.503,E2 -18329.503} C_VEL
LIN {X 0,Y 263.144,Z 651.832,A -85,B 0,C 180,E1 -18332.997,E2 -18332.997} C_VEL
LIN {X 0,Y 263.147,Z 651.814,A -85,B 0,C 180,E1 -18336.383,E2 -18336.383} C_VEL
LIN {X 0,Y 263.24,Z 651.818,A -85,B 0,C 180,E1 -18339.691,E2 -18339.691} C_VEL
LIN {X 0,Y 263.206,Z 651.81,A -85,B 0,C 180,E1 -18340.829,E2 -18340.829} C_VEL
LIN {X 0,Y 262.57,Z 651.888,A -85,B 0,C 180,E1 -18342.106,E2 -18342.106} C_VEL
LIN {X 0,Y 259.77,Z 652.249,A -85,B 0,C 180,E1 -18344.189,E2 -18344.189} C_VEL
LIN {X 0,Y 257.376,Z 652.552,A -85,B 0,C 180,E1 -18345.883,E2 -18345.883} C_VEL
LIN {X 0,Y 256.34,Z 652.675,A -85,B 0,C 180,E1 -18347.196,E2 -18347.196} C_VEL
LIN {X 0,Y 256.253,Z 652.68,A -85,B 0,C 180,E1 -18347.641,E2 -18347.641} C_VEL
LIN {X 0,Y 256.436,Z 652.65,A -85,B 0,C 180,E1 -18350.622,E2 -18350.622} C_VEL
LIN {X 0,Y 256.461,Z 652.665,A -85,B 0,C 180,E1 -18353.706,E2 -18353.706} C_VEL
LIN {X 0,Y 256.714,Z 652.632,A -85,B 0,C 180,E1 -18358.431,E2 -18358.431} C_VEL
LIN {X 0,Y 256.715,Z 652.623,A -85,B 0,C 180,E1 -18361.568,E2 -18361.568} C_VEL
LIN {X 0,Y 256.482,Z 652.653,A -85,B 0,C 180,E1 -18366.292,E2 -18366.292} C_VEL
LIN {X 0,Y 256.429,Z 652.666,A -85,B 0,C 180,E1 -18369.464,E2 -18369.464} C_VEL
LIN {X 0,Y 256.258,Z 652.683,A -85,B 0,C 180,E1 -18374.29,E2 -18374.29} C_VEL
LIN {X 0,Y 256.213,Z 652.692,A -85,B 0,C 180,E1 -18377.561,E2 -18377.561} C_VEL
LIN {X 0,Y 256.155,Z 652.698,A -85,B 0,C 180,E1 -18381.117,E2 -18381.117} C_VEL
LIN {X 0,Y 256.172,Z 652.697,A -85,B 0,C 180,E1 -18385.13,E2 -18385.13} C_VEL
LIN {X 0,Y 256.115,Z 652.706,A -85,B 0,C 180,E1 -18389.599,E2 -18389.599} C_VEL
LIN {X 0,Y 256.086,Z 652.709,A -85,B 0,C 180,E1 -18393.29,E2 -18393.29} C_VEL
LIN {X 0,Y 256.141,Z 652.701,A -85,B 0,C 180,E1 -18397.278,E2 -18397.278} C_VEL
LIN {X 0,Y 256.085,Z 652.709,A -85,B 0,C 180,E1 -18401.197,E2 -18401.197} C_VEL
LIN {X 0,Y 256.069,Z 652.71,A -85,B 0,C 180,E1 -18404.472,E2 -18404.472} C_VEL
LIN {X 0,Y 256.1,Z 652.87,A -85,B 0,C 180,E1 -18407.65,E2 -18407.65} C_VEL
LIN {X 0,Y 258.732,Z 662.257,A -85,B 0,C 180,E1 -18411.336,E2 -18411.336} C_VEL
LIN {X 0,Y 259.556,Z 665.504,A -85,B 0,C 180,E1 -18412.517,E2 -18412.517} C_VEL
LIN {X 0,Y 268.55,Z 684.825,A -85,B 0,C 180,E1 -18414.459,E2 -18414.459} C_VEL
LIN {X 0,Y 275.097,Z 700.863,A -85,B 0,C 180,E1 -18415.827,E2 -18415.827} C_VEL
LIN {X 0,Y 278.069,Z 722.531,A -85,B 0,C 180,E1 -18416.846,E2 -18416.846} C_VEL
LIN {X 0,Y 275.085,Z 803.433,A -85,B 0,C 180,E1 -18418.898,E2 -18418.898} C_VEL
LIN {X 0,Y 273.903,Z 817.704,A -85,B 0,C 180,E1 -18419.498,E2 -18419.498} C_VEL
LIN {X 0,Y 272.238,Z 832.06,A -85,B 0,C 180,E1 -18420.414,E2 -18420.414} C_VEL
LIN {X 0,Y 270.329,Z 844.401,A -85,B 0,C 180,E1 -18421.464,E2 -18421.464} C_VEL
LIN {X 0,Y 268.228,Z 856.498,A -85,B 0,C 180,E1 -18422.792,E2 -18422.792} C_VEL
LIN {X 0,Y 265.919,Z 868.102,A -85,B 0,C 180,E1 -18424.384,E2 -18424.384} C_VEL
LIN {X 0,Y 263.783,Z 877.93,A -85,B 0,C 180,E1 -18426.027,E2 -18426.027} C_VEL
LIN {X 0,Y 261.592,Z 887.277,A -85,B 0,C 180,E1 -18427.906,E2 -18427.906} C_VEL
LIN {X 0,Y 259.463,Z 896.642,A -85,B 0,C 180,E1 -18430.209,E2 -18430.209} C_VEL
LIN {X 0,Y 257.41,Z 905.372,A -85,B 0,C 180,E1 -18432.861,E2 -18432.861} C_VEL
LIN {X 0,Y 256.352,Z 910.916,A -85,B 0,C 180,E1 -18434.903,E2 -18434.903} C_VEL
LIN {X 0,Y 255.277,Z 916.258,A -85,B 0,C 180,E1 -18437.276,E2 -18437.276} C_VEL
LIN {X 0,Y 254.448,Z 921.895,A -85,B 0,C 180,E1 -18440.461,E2 -18440.461} C_VEL
LIN {X 0,Y 254.068,Z 925.947,A -85,B 0,C 180,E1 -18443.647,E2 -18443.647} C_VEL
LIN {X 0,Y 254.052,Z 928.528,A -85,B 0,C 180,E1 -18446.828,E2 -18446.828} C_VEL
LIN {X 0,Y 254.102,Z 929.723,A -85,B 0,C 180,E1 -18450,E2 -18450} C_VEL
LIN {X 0,Y 254.075,Z 929.811,A -85,B 0,C 180,E1 -18451.585,E2 -18451.585} C_VEL
LIN {X 0,Y 254.012,Z 928.978,A -85,B 0,C 180,E1 -18454.761,E2 -18454.761} C_VEL
LIN {X 0,Y 254.22,Z 926.801,A -85,B 0,C 180,E1 -18457.945,E2 -18457.945} C_VEL
LIN {X 0,Y 254.854,Z 923.232,A -85,B 0,C 180,E1 -18461.13,E2 -18461.13} C_VEL
LIN {X 0,Y 256.176,Z 918.176,A -85,B 0,C 180,E1 -18464.295,E2 -18464.295} C_VEL
LIN {X 0,Y 258.123,Z 911.49,A -85,B 0,C 180,E1 -18467.427,E2 -18467.427} C_VEL
LIN {X 0,Y 260.282,Z 904.068,A -85,B 0,C 180,E1 -18470.137,E2 -18470.137} C_VEL
LIN {X 0,Y 263.111,Z 894.87,A -85,B 0,C 180,E1 -18472.787,E2 -18472.787} C_VEL
LIN {X 0,Y 266.039,Z 885.281,A -85,B 0,C 180,E1 -18475.003,E2 -18475.003} C_VEL
LIN {X 0,Y 269.342,Z 873.929,A -85,B 0,C 180,E1 -18477.106,E2 -18477.106} C_VEL
LIN {X 0,Y 271.896,Z 863.357,A -85,B 0,C 180,E1 -18478.715,E2 -18478.715} C_VEL
LIN {X 0,Y 274.636,Z 851.549,A -85,B 0,C 180,E1 -18480.146,E2 -18480.146} C_VEL
LIN {X 0,Y 277.159,Z 839.18,A -85,B 0,C 180,E1 -18481.32,E2 -18481.32} C_VEL
LIN {X 0,Y 279.354,Z 825.487,A -85,B 0,C 180,E1 -18482.317,E2 -18482.317} C_VEL
LIN {X 0,Y 281.111,Z 811.237,A -85,B 0,C 180,E1 -18483.047,E2 -18483.047} C_VEL
LIN {X 0,Y 282.135,Z 796.91,A -85,B 0,C 180,E1 -18483.521,E2 -18483.521} C_VEL
LIN {X 0,Y 285.126,Z 723.901,A -85,B 0,C 180,E1 -18485.327,E2 -18485.327} C_VEL
LIN {X 0,Y 282.902,Z 710.307,A -85,B 0,C 180,E1 -18486.098,E2 -18486.098} C_VEL
LIN {X 0,Y 275.86,Z 694.589,A -85,B 0,C 180,E1 -18487.769,E2 -18487.769} C_VEL
LIN {X 0,Y 270.198,Z 683.307,A -85,B 0,C 180,E1 -18489.161,E2 -18489.161} C_VEL
LIN {X 0,Y 264.563,Z 673.191,A -85,B 0,C 180,E1 -18490.599,E2 -18490.599} C_VEL
LIN {X 0,Y 261.927,Z 668.655,A -85,B 0,C 180,E1 -18491.298,E2 -18491.298} C_VEL
LIN {X 0,Y 259.649,Z 664.481,A -85,B 0,C 180,E1 -18491.971,E2 -18491.971} C_VEL
LIN {X 0,Y 257.091,Z 656.144,A -85,B 0,C 180,E1 -18495.753,E2 -18495.753} C_VEL
LIN {X 0,Y 256.079,Z 652.693,A -85,B 0,C 180,E1 -18497.47,E2 -18497.47} C_VEL
LIN {X 0,Y 256.1,Z 652.701,A -85,B 0,C 180,E1 -18500.864,E2 -18500.864} C_VEL
LIN {X 0,Y 256.121,Z 652.702,A -85,B 0,C 180,E1 -18504.814,E2 -18504.814} C_VEL
LIN {X 0,Y 256.092,Z 652.675,A -85,B 0,C 180,E1 -18508.573,E2 -18508.573} C_VEL
LIN {X 0,Y 256.143,Z 652.701,A -85,B 0,C 180,E1 -18512.197,E2 -18512.197} C_VEL
LIN {X 0,Y 256.173,Z 652.7,A -85,B 0,C 180,E1 -18515.7,E2 -18515.7} C_VEL
LIN {X 0,Y 256.168,Z 652.698,A -85,B 0,C 180,E1 -18519.105,E2 -18519.105} C_VEL
LIN {X 0,Y 256.301,Z 652.686,A -85,B 0,C 180,E1 -18524.086,E2 -18524.086} C_VEL
LIN {X 0,Y 256.298,Z 652.684,A -85,B 0,C 180,E1 -18528.934,E2 -18528.934} C_VEL
LIN {X 0,Y 256.516,Z 652.65,A -85,B 0,C 180,E1 -18532.127,E2 -18532.127} C_VEL
LIN {X 0,Y 256.499,Z 652.652,A -85,B 0,C 180,E1 -18536.859,E2 -18536.859} C_VEL
LIN {X 0,Y 256.759,Z 652.616,A -85,B 0,C 180,E1 -18540,E2 -18540} C_VEL
LIN {X 0,Y 256.5,Z 652.659,A -85,B 0,C 180,E1 -18543.142,E2 -18543.142} C_VEL
LIN {X 0,Y 256.517,Z 652.657,A -85,B 0,C 180,E1 -18547.874,E2 -18547.874} C_VEL
LIN {X 0,Y 256.297,Z 652.687,A -85,B 0,C 180,E1 -18552.673,E2 -18552.673} C_VEL
LIN {X 0,Y 256.284,Z 652.681,A -85,B 0,C 180,E1 -18556.303,E2 -18556.303} C_VEL
LIN {X 0,Y 256.155,Z 652.702,A -85,B 0,C 180,E1 -18561.118,E2 -18561.118} C_VEL
LIN {X 0,Y 256.162,Z 652.701,A -85,B 0,C 180,E1 -18565.126,E2 -18565.126} C_VEL
LIN {X 0,Y 256.057,Z 652.68,A -85,B 0,C 180,E1 -18569.608,E2 -18569.608} C_VEL
LIN {X 0,Y 256.068,Z 652.709,A -85,B 0,C 180,E1 -18573.293,E2 -18573.293} C_VEL
LIN {X 0,Y 256.111,Z 652.703,A -85,B 0,C 180,E1 -18577.27,E2 -18577.27} C_VEL
LIN {X 0,Y 256.059,Z 652.701,A -85,B 0,C 180,E1 -18582.178,E2 -18582.178} C_VEL
LIN {X 0,Y 256.035,Z 652.722,A -85,B 0,C 180,E1 -18582.409,E2 -18582.409} C_VEL
LIN {X 0,Y 256.995,Z 655.497,A -85,B 0,C 180,E1 -18582.731,E2 -18582.731} C_VEL
LIN {X 0,Y 259.26,Z 658.208,A -85,B 0,C 180,E1 -18583.329,E2 -18583.329} C_VEL
LIN {X 0,Y 261.569,Z 661.628,A -85,B 0,C 180,E1 -18583.946,E2 -18583.946} C_VEL
LIN {X 0,Y 269.966,Z 674.334,A -85,B 0,C 180,E1 -18586.062,E2 -18586.062} C_VEL
LIN {X 0,Y 274.402,Z 681.785,A -85,B 0,C 180,E1 -18587.126,E2 -18587.126} C_VEL
LIN {X 0,Y 281.758,Z 696.235,A -85,B 0,C 180,E1 -18588.85,E2 -18588.85} C_VEL
LIN {X 0,Y 285.864,Z 705.402,A -85,B 0,C 180,E1 -18589.79,E2 -18589.79} C_VEL
LIN {X 0,Y 282.453,Z 786.165,A -85,B 0,C 180,E1 -18591.818,E2 -18591.818} C_VEL
LIN {X 0,Y 281.133,Z 800.879,A -85,B 0,C 180,E1 -18592.458,E2 -18592.458} C_VEL
LIN {X 0,Y 279.294,Z 814.781,A -85,B 0,C 180,E1 -18593.344,E2 -18593.344} C_VEL
LIN {X 0,Y 277.227,Z 826.567,A -85,B 0,C 180,E1 -18594.333,E2 -18594.333} C_VEL
LIN {X 0,Y 274.678,Z 839.424,A -85,B 0,C 180,E1 -18595.743,E2 -18595.743} C_VEL
LIN {X 0,Y 271.96,Z 851.073,A -85,B 0,C 180,E1 -18597.354,E2 -18597.354} C_VEL
LIN {X 0,Y 269.386,Z 860.742,A -85,B 0,C 180,E1 -18598.986,E2 -18598.986} C_VEL
LIN {X 0,Y 266.408,Z 871.436,A -85,B 0,C 180,E1 -18601.22,E2 -18601.22} C_VEL
LIN {X 0,Y 263.658,Z 880.233,A -85,B 0,C 180,E1 -18603.482,E2 -18603.482} C_VEL
LIN {X 0,Y 261.274,Z 887.523,A -85,B 0,C 180,E1 -18605.782,E2 -18605.782} C_VEL
LIN {X 0,Y 259.027,Z 894.47,A -85,B 0,C 180,E1 -18608.513,E2 -18608.513} C_VEL
LIN {X 0,Y 256.97,Z 900.677,A -85,B 0,C 180,E1 -18611.668,E2 -18611.668} C_VEL
LIN {X 0,Y 255.892,Z 904.19,A -85,B 0,C 180,E1 -18614.059,E2 -18614.059} C_VEL
LIN {X 0,Y 254.791,Z 907.61,A -85,B 0,C 180,E1 -18617.252,E2 -18617.252} C_VEL
LIN {X 0,Y 254.264,Z 909.626,A -85,B 0,C 180,E1 -18620.454,E2 -18620.454} C_VEL
LIN {X 0,Y 254.139,Z 910.303,A -85,B 0,C 180,E1 -18623.649,E2 -18623.649} C_VEL
LIN {X 0,Y 254.104,Z 909.668,A -85,B 0,C 180,E1 -18626.829,E2 -18626.829} C_VEL
LIN {X 0,Y 254.204,Z 907.713,A -85,B 0,C 180,E1 -18630,E2 -18630} C_VEL
LIN {X 0,Y 254.645,Z 904.391,A -85,B 0,C 180,E1 -18633.164,E2 -18633.164} C_VEL
LIN {X 0,Y 255.67,Z 899.598,A -85,B 0,C 180,E1 -18636.313,E2 -18636.313} C_VEL
LIN {X 0,Y 256.741,Z 894.981,A -85,B 0,C 180,E1 -18638.659,E2 -18638.659} C_VEL
LIN {X 0,Y 258.317,Z 888.441,A -85,B 0,C 180,E1 -18641.315,E2 -18641.315} C_VEL
LIN {X 0,Y 259.847,Z 881.29,A -85,B 0,C 180,E1 -18643.69,E2 -18643.69} C_VEL
LIN {X 0,Y 262.043,Z 872.86,A -85,B 0,C 180,E1 -18645.957,E2 -18645.957} C_VEL
LIN {X 0,Y 264.491,Z 862.668,A -85,B 0,C 180,E1 -18648.193,E2 -18648.193} C_VEL
LIN {X 0,Y 266.811,Z 851.293,A -85,B 0,C 180,E1 -18650.226,E2 -18650.226} C_VEL
LIN {X 0,Y 269.176,Z 838.545,A -85,B 0,C 180,E1 -18652.044,E2 -18652.044} C_VEL
LIN {X 0,Y 271.365,Z 825.773,A -85,B 0,C 180,E1 -18653.465,E2 -18653.465} C_VEL
LIN {X 0,Y 273.195,Z 812.496,A -85,B 0,C 180,E1 -18654.609,E2 -18654.609} C_VEL
LIN {X 0,Y 274.595,Z 798.765,A -85,B 0,C 180,E1 -18655.487,E2 -18655.487} C_VEL
LIN {X 0,Y 275.496,Z 785.308,A -85,B 0,C 180,E1 -18656.075,E2 -18656.075} C_VEL
LIN {X 0,Y 278.835,Z 699.436,A -85,B 0,C 180,E1 -18658.234,E2 -18658.234} C_VEL
LIN {X 0,Y 274.701,Z 688.713,A -85,B 0,C 180,E1 -18659.085,E2 -18659.085} C_VEL
LIN {X 0,Y 268.124,Z 674.366,A -85,B 0,C 180,E1 -18660.423,E2 -18660.423} C_VEL
LIN {X 0,Y 260.17,Z 660.401,A -85,B 0,C 180,E1 -18662.05,E2 -18662.05} C_VEL
LIN {X 0,Y 257.64,Z 656.318,A -85,B 0,C 180,E1 -18662.584,E2 -18662.584} C_VEL
LIN {X 0,Y 256.319,Z 653.882,A -85,B 0,C 180,E1 -18662.878,E2 -18662.878} C_VEL
LIN {X 0,Y 256.079,Z 652.712,A -85,B 0,C 180,E1 -18663.01,E2 -18663.01} C_VEL
LIN {X 0,Y 256.089,Z 652.712,A -85,B 0,C 180,E1 -18667.262,E2 -18667.262} C_VEL
LIN {X 0,Y 256.065,Z 652.713,A -85,B 0,C 180,E1 -18672.178,E2 -18672.178} C_VEL
LIN {X 0,Y 256.037,Z 652.713,A -85,B 0,C 180,E1 -18676.667,E2 -18676.667} C_VEL
LIN {X 0,Y 256.044,Z 652.698,A -85,B 0,C 180,E1 -18680.852,E2 -18680.852} C_VEL
LIN {X 0,Y 256.08,Z 652.696,A -85,B 0,C 180,E1 -18684.806,E2 -18684.806} C_VEL
LIN {X 0,Y 256.085,Z 652.703,A -85,B 0,C 180,E1 -18688.571,E2 -18688.571} C_VEL
LIN {X 0,Y 256.096,Z 652.708,A -85,B 0,C 180,E1 -18692.19,E2 -18692.19} C_VEL
LIN {X 0,Y 256.135,Z 652.686,A -85,B 0,C 180,E1 -18695.695,E2 -18695.695} C_VEL
LIN {X 0,Y 256.149,Z 652.703,A -85,B 0,C 180,E1 -18699.103,E2 -18699.103} C_VEL
LIN {X 0,Y 256.251,Z 652.679,A -85,B 0,C 180,E1 -18704.081,E2 -18704.081} C_VEL
LIN {X 0,Y 256.253,Z 652.68,A -85,B 0,C 180,E1 -18707.641,E2 -18707.641} C_VEL
LIN {X 0,Y 255.6,Z 652.753,A -85,B 0,C 180,E1 -18708.955,E2 -18708.955} C_VEL
LIN {X 0,Y 252.838,Z 653.103,A -85,B 0,C 180,E1 -18711.1,E2 -18711.1} C_VEL
LIN {X 0,Y 249.658,Z 653.512,A -85,B 0,C 180,E1 -18713.741,E2 -18713.741} C_VEL
LIN {X 0,Y 249.307,Z 653.548,A -85,B 0,C 180,E1 -18714.654,E2 -18714.654} C_VEL
LIN {X 0,Y 249.675,Z 653.509,A -85,B 0,C 180,E1 -18718.387,E2 -18718.387} C_VEL
LIN {X 0,Y 249.677,Z 653.5,A -85,B 0,C 180,E1 -18721.613,E2 -18721.613} C_VEL
LIN {X 0,Y 249.454,Z 653.529,A -85,B 0,C 180,E1 -18726.47,E2 -18726.47} C_VEL
LIN {X 0,Y 249.345,Z 653.545,A -85,B 0,C 180,E1 -18729.736,E2 -18729.736} C_VEL
LIN {X 0,Y 249.208,Z 653.559,A -85,B 0,C 180,E1 -18734.703,E2 -18734.703} C_VEL
LIN {X 0,Y 249.141,Z 653.573,A -85,B 0,C 180,E1 -18738.077,E2 -18738.077} C_VEL
LIN {X 0,Y 249.086,Z 653.579,A -85,B 0,C 180,E1 -18741.518,E2 -18741.518} C_VEL
LIN {X 0,Y 249.119,Z 653.576,A -85,B 0,C 180,E1 -18745.475,E2 -18745.475} C_VEL
LIN {X 0,Y 249.085,Z 653.582,A -85,B 0,C 180,E1 -18748.993,E2 -18748.993} C_VEL
LIN {X 0,Y 249.037,Z 653.591,A -85,B 0,C 180,E1 -18752.424,E2 -18752.424} C_VEL
LIN {X 0,Y 249.076,Z 653.582,A -85,B 0,C 180,E1 -18756.337,E2 -18756.337} C_VEL
LIN {X 0,Y 249.045,Z 653.588,A -85,B 0,C 180,E1 -18760.47,E2 -18760.47} C_VEL
LIN {X 0,Y 249.013,Z 653.591,A -85,B 0,C 180,E1 -18764.876,E2 -18764.876} C_VEL
LIN {X 0,Y 249.062,Z 653.678,A -85,B 0,C 180,E1 -18766.702,E2 -18766.702} C_VEL
LIN {X 0,Y 252.214,Z 665.114,A -85,B 0,C 180,E1 -18771.327,E2 -18771.327} C_VEL
LIN {X 0,Y 260.983,Z 683.404,A -85,B 0,C 180,E1 -18773.323,E2 -18773.323} C_VEL
LIN {X 0,Y 268.858,Z 702.125,A -85,B 0,C 180,E1 -18775.04,E2 -18775.04} C_VEL
LIN {X 0,Y 269.907,Z 707.596,A -85,B 0,C 180,E1 -18775.351,E2 -18775.351} C_VEL
LIN {X 0,Y 271.981,Z 723.867,A -85,B 0,C 180,E1 -18776.121,E2 -18776.121} C_VEL
LIN {X 0,Y 268.833,Z 804.17,A -85,B 0,C 180,E1 -18778.201,E2 -18778.201} C_VEL
LIN {X 0,Y 267.508,Z 818.802,A -85,B 0,C 180,E1 -18778.853,E2 -18778.853} C_VEL
LIN {X 0,Y 265.721,Z 833.374,A -85,B 0,C 180,E1 -18779.832,E2 -18779.832} C_VEL
LIN {X 0,Y 263.762,Z 845.371,A -85,B 0,C 180,E1 -18780.904,E2 -18780.904} C_VEL
LIN {X 0,Y 261.429,Z 858.094,A -85,B 0,C 180,E1 -18782.372,E2 -18782.372} C_VEL
LIN {X 0,Y 259.17,Z 868.884,A -85,B 0,C 180,E1 -18783.924,E2 -18783.924} C_VEL
LIN {X 0,Y 256.777,Z 879.332,A -85,B 0,C 180,E1 -18785.76,E2 -18785.76} C_VEL
LIN {X 0,Y 254.57,Z 888.406,A -85,B 0,C 180,E1 -18787.691,E2 -18787.691} C_VEL
LIN {X 0,Y 252.38,Z 897.533,A -85,B 0,C 180,E1 -18790.054,E2 -18790.054} C_VEL
LIN {X 0,Y 250.2,Z 906.494,A -85,B 0,C 180,E1 -18792.935,E2 -18792.935} C_VEL
LIN {X 0,Y 249.051,Z 912.389,A -85,B 0,C 180,E1 -18795.287,E2 -18795.287} C_VEL
LIN {X 0,Y 247.752,Z 918.901,A -85,B 0,C 180,E1 -18798.546,E2 -18798.546} C_VEL
LIN {X 0,Y 247.161,Z 923.758,A -85,B 0,C 180,E1 -18801.826,E2 -18801.826} C_VEL
LIN {X 0,Y 246.969,Z 927.096,A -85,B 0,C 180,E1 -18805.102,E2 -18805.102} C_VEL
LIN {X 0,Y 247.013,Z 929.006,A -85,B 0,C 180,E1 -18808.369,E2 -18808.369} C_VEL
LIN {X 0,Y 247.029,Z 929.445,A -85,B 0,C 180,E1 -18810,E2 -18810} C_VEL
LIN {X 0,Y 247.003,Z 929.545,A -85,B 0,C 180,E1 -18811.63,E2 -18811.63} C_VEL
LIN {X 0,Y 246.95,Z 928.642,A -85,B 0,C 180,E1 -18815.081,E2 -18815.081} C_VEL
LIN {X 0,Y 247.158,Z 926.581,A -85,B 0,C 180,E1 -18818.174,E2 -18818.174} C_VEL
LIN {X 0,Y 247.85,Z 923.036,A -85,B 0,C 180,E1 -18821.449,E2 -18821.449} C_VEL
LIN {X 0,Y 249.267,Z 918.007,A -85,B 0,C 180,E1 -18824.7,E2 -18824.7} C_VEL
LIN {X 0,Y 251.268,Z 911.349,A -85,B 0,C 180,E1 -18827.919,E2 -18827.919} C_VEL
LIN {X 0,Y 253.578,Z 903.966,A -85,B 0,C 180,E1 -18830.693,E2 -18830.693} C_VEL
LIN {X 0,Y 256.551,Z 894.819,A -85,B 0,C 180,E1 -18833.404,E2 -18833.404} C_VEL
LIN {X 0,Y 259.609,Z 885.276,A -85,B 0,C 180,E1 -18835.667,E2 -18835.667} C_VEL
LIN {X 0,Y 262.93,Z 874.353,A -85,B 0,C 180,E1 -18837.748,E2 -18837.748} C_VEL
LIN {X 0,Y 265.694,Z 863.475,A -85,B 0,C 180,E1 -18839.45,E2 -18839.45} C_VEL
LIN {X 0,Y 268.525,Z 851.756,A -85,B 0,C 180,E1 -18840.906,E2 -18840.906} C_VEL
LIN {X 0,Y 271.144,Z 839.509,A -85,B 0,C 180,E1 -18842.097,E2 -18842.097} C_VEL
LIN {X 0,Y 273.411,Z 826.001,A -85,B 0,C 180,E1 -18843.109,E2 -18843.109} C_VEL
LIN {X 0,Y 275.23,Z 812.07,A -85,B 0,C 180,E1 -18843.847,E2 -18843.847} C_VEL
LIN {X 0,Y 276.367,Z 797.369,A -85,B 0,C 180,E1 -18844.358,E2 -18844.358} C_VEL
LIN {X 0,Y 279.467,Z 725.042,A -85,B 0,C 180,E1 -18846.177,E2 -18846.177} C_VEL
LIN {X 0,Y 277.603,Z 713.339,A -85,B 0,C 180,E1 -18846.858,E2 -18846.858} C_VEL
LIN {X 0,Y 269.49,Z 695.183,A -85,B 0,C 180,E1 -18848.882,E2 -18848.882} C_VEL
LIN {X 0,Y 262.73,Z 682.283,A -85,B 0,C 180,E1 -18850.635,E2 -18850.635} C_VEL
LIN {X 0,Y 257.475,Z 673.043,A -85,B 0,C 180,E1 -18852.07,E2 -18852.07} C_VEL
LIN {X 0,Y 254.746,Z 668.533,A -85,B 0,C 180,E1 -18852.842,E2 -18852.842} C_VEL
LIN {X 0,Y 252.267,Z 664.191,A -85,B 0,C 180,E1 -18853.586,E2 -18853.586} C_VEL
LIN {X 0,Y 249.794,Z 656.015,A -85,B 0,C 180,E1 -18857.527,E2 -18857.527} C_VEL
LIN {X 0,Y 249.055,Z 653.571,A -85,B 0,C 180,E1 -18858.865,E2 -18858.865} C_VEL
LIN {X 0,Y 249.074,Z 653.563,A -85,B 0,C 180,E1 -18863.662,E2 -18863.662} C_VEL
LIN {X 0,Y 249.04,Z 653.556,A -85,B 0,C 180,E1 -18867.845,E2 -18867.845} C_VEL
LIN {X 0,Y 249.097,Z 653.577,A -85,B 0,C 180,E1 -18871.339,E2 -18871.339} C_VEL
LIN {X 0,Y 249.156,Z 653.57,A -85,B 0,C 180,E1 -18874.969,E2 -18874.969} C_VEL
LIN {X 0,Y 249.112,Z 653.577,A -85,B 0,C 180,E1 -18880.212,E2 -18880.212} C_VEL
LIN {X 0,Y 249.242,Z 653.562,A -85,B 0,C 180,E1 -18883.622,E2 -18883.622} C_VEL
LIN {X 0,Y 249.246,Z 653.563,A -85,B 0,C 180,E1 -18888.617,E2 -18888.617} C_VEL
LIN {X 0,Y 249.456,Z 653.527,A -85,B 0,C 180,E1 -18891.902,E2 -18891.902} C_VEL
LIN {X 0,Y 249.297,Z 653.544,A -85,B 0,C 180,E1 -18895.149,E2 -18895.149} C_VEL
LIN {X 0,Y 249.677,Z 653.51,A -85,B 0,C 180,E1 -18898.387,E2 -18898.387} C_VEL
LIN {X 0,Y 249.677,Z 653.5,A -85,B 0,C 180,E1 -18901.613,E2 -18901.613} C_VEL
LIN {X 0,Y 249.443,Z 653.527,A -85,B 0,C 180,E1 -18906.712,E2 -18906.712} C_VEL
LIN {X 0,Y 249.345,Z 653.54,A -85,B 0,C 180,E1 -18909.737,E2 -18909.737} C_VEL
LIN {X 0,Y 249.207,Z 653.556,A -85,B 0,C 180,E1 -18914.704,E2 -18914.704} C_VEL
LIN {X 0,Y 249.14,Z 653.573,A -85,B 0,C 180,E1 -18918.078,E2 -18918.078} C_VEL
LIN {X 0,Y 249.085,Z 653.583,A -85,B 0,C 180,E1 -18921.519,E2 -18921.519} C_VEL
LIN {X 0,Y 249.107,Z 653.581,A -85,B 0,C 180,E1 -18925.47,E2 -18925.47} C_VEL
LIN {X 0,Y 249.04,Z 653.552,A -85,B 0,C 180,E1 -18928.975,E2 -18928.975} C_VEL
LIN {X 0,Y 249.029,Z 653.591,A -85,B 0,C 180,E1 -18932.427,E2 -18932.427} C_VEL
LIN {X 0,Y 249.028,Z 653.586,A -85,B 0,C 180,E1 -18936.346,E2 -18936.346} C_VEL
LIN {X 0,Y 248.986,Z 653.573,A -85,B 0,C 180,E1 -18940.782,E2 -18940.782} C_VEL
LIN {X 0,Y 249.99,Z 656.413,A -85,B 0,C 180,E1 -18941.15,E2 -18941.15} C_VEL
LIN {X 0,Y 252.202,Z 658.872,A -85,B 0,C 180,E1 -18941.774,E2 -18941.774} C_VEL
LIN {X 0,Y 254.286,Z 662.209,A -85,B 0,C 180,E1 -18942.386,E2 -18942.386} C_VEL
LIN {X 0,Y 255.925,Z 664.449,A -85,B 0,C 180,E1 -18942.84,E2 -18942.84} C_VEL
LIN {X 0,Y 261.363,Z 672.413,A -85,B 0,C 180,E1 -18944.303,E2 -18944.303} C_VEL
LIN {X 0,Y 269.08,Z 684.733,A -85,B 0,C 180,E1 -18946.258,E2 -18946.258} C_VEL
LIN {X 0,Y 276.849,Z 700.104,A -85,B 0,C 180,E1 -18948.161,E2 -18948.161} C_VEL
LIN {X 0,Y 280.157,Z 707.529,A -85,B 0,C 180,E1 -18948.951,E2 -18948.951} C_VEL
LIN {X 0,Y 276.766,Z 785.693,A -85,B 0,C 180,E1 -18950.945,E2 -18950.945} C_VEL
LIN {X 0,Y 275.479,Z 799.938,A -85,B 0,C 180,E1 -18951.548,E2 -18951.548} C_VEL
LIN {X 0,Y 273.612,Z 814.159,A -85,B 0,C 180,E1 -18952.454,E2 -18952.454} C_VEL
LIN {X 0,Y 271.429,Z 826.138,A -85,B 0,C 180,E1 -18953.45,E2 -18953.45} C_VEL
LIN {X 0,Y 268.772,Z 839.131,A -85,B 0,C 180,E1 -18954.882,E2 -18954.882} C_VEL
LIN {X 0,Y 265.891,Z 850.879,A -85,B 0,C 180,E1 -18956.512,E2 -18956.512} C_VEL
LIN {X 0,Y 263.228,Z 860.628,A -85,B 0,C 180,E1 -18958.177,E2 -18958.177} C_VEL
LIN {X 0,Y 260.594,Z 869.902,A -85,B 0,C 180,E1 -18960.111,E2 -18960.111} C_VEL
LIN {X 0,Y 257.67,Z 878.882,A -85,B 0,C 180,E1 -18962.375,E2 -18962.375} C_VEL
LIN {X 0,Y 254.699,Z 887.576,A -85,B 0,C 180,E1 -18965.115,E2 -18965.115} C_VEL
LIN {X 0,Y 252.339,Z 894.564,A -85,B 0,C 180,E1 -18967.914,E2 -18967.914} C_VEL
LIN {X 0,Y 250.148,Z 900.812,A -85,B 0,C 180,E1 -18971.15,E2 -18971.15} C_VEL
LIN {X 0,Y 248.927,Z 904.518,A -85,B 0,C 180,E1 -18973.728,E2 -18973.728} C_VEL
LIN {X 0,Y 247.786,Z 907.813,A -85,B 0,C 180,E1 -18976.885,E2 -18976.885} C_VEL
LIN {X 0,Y 247.207,Z 909.861,A -85,B 0,C 180,E1 -18980.179,E2 -18980.179} C_VEL
LIN {X 0,Y 247.043,Z 910.57,A -85,B 0,C 180,E1 -18983.466,E2 -18983.466} C_VEL
LIN {X 0,Y 247.018,Z 909.971,A -85,B 0,C 180,E1 -18986.738,E2 -18986.738} C_VEL
LIN {X 0,Y 247.126,Z 908.056,A -85,B 0,C 180,E1 -18990,E2 -18990} C_VEL
LIN {X 0,Y 247.578,Z 904.769,A -85,B 0,C 180,E1 -18993.255,E2 -18993.255} C_VEL
LIN {X 0,Y 248.641,Z 900.012,A -85,B 0,C 180,E1 -18996.492,E2 -18996.492} C_VEL
LIN {X 0,Y 249.755,Z 895.43,A -85,B 0,C 180,E1 -18998.903,E2 -18998.903} C_VEL
LIN {X 0,Y 251.482,Z 888.507,A -85,B 0,C 180,E1 -19001.786,E2 -19001.786} C_VEL
LIN {X 0,Y 252.973,Z 881.815,A -85,B 0,C 180,E1 -19004.069,E2 -19004.069} C_VEL
LIN {X 0,Y 255.256,Z 873.432,A -85,B 0,C 180,E1 -19006.393,E2 -19006.393} C_VEL
LIN {X 0,Y 257.783,Z 863.326,A -85,B 0,C 180,E1 -19008.684,E2 -19008.684} C_VEL
LIN {X 0,Y 260.197,Z 852.028,A -85,B 0,C 180,E1 -19010.764,E2 -19010.764} C_VEL
LIN {X 0,Y 262.363,Z 840.794,A -85,B 0,C 180,E1 -19012.44,E2 -19012.44} C_VEL
LIN {X 0,Y 264.62,Z 828.489,A -85,B 0,C 180,E1 -19013.893,E2 -19013.893} C_VEL
LIN {X 0,Y 266.698,Z 814.765,A -85,B 0,C 180,E1 -19015.146,E2 -19015.146} C_VEL
LIN {X 0,Y 268.2,Z 801,A -85,B 0,C 180,E1 -19016.088,E2 -19016.088} C_VEL
LIN {X 0,Y 269.202,Z 787.227,A -85,B 0,C 180,E1 -19016.741,E2 -19016.741} C_VEL
LIN {X 0,Y 270.845,Z 749.32,A -85,B 0,C 180,E1 -19017.746,E2 -19017.746} C_VEL
LIN {X 0,Y 272.631,Z 700.674,A -85,B 0,C 180,E1 -19018.993,E2 -19018.993} C_VEL
LIN {X 0,Y 265.608,Z 683.777,A -85,B 0,C 180,E1 -19020.483,E2 -19020.483} C_VEL
LIN {X 0,Y 260.846,Z 674.431,A -85,B 0,C 180,E1 -19021.485,E2 -19021.485} C_VEL
LIN {X 0,Y 252.974,Z 661.011,A -85,B 0,C 180,E1 -19023.183,E2 -19023.183} C_VEL
LIN {X 0,Y 250.686,Z 657.306,A -85,B 0,C 180,E1 -19023.696,E2 -19023.696} C_VEL
LIN {X 0,Y 249.314,Z 654.855,A -85,B 0,C 180,E1 -19024.018,E2 -19024.018} C_VEL
LIN {X 0,Y 249.055,Z 653.586,A -85,B 0,C 180,E1 -19024.139,E2 -19024.139} C_VEL
LIN {X 0,Y 249.005,Z 653.584,A -85,B 0,C 180,E1 -19028.385,E2 -19028.385} C_VEL
LIN {X 0,Y 248.999,Z 653.594,A -85,B 0,C 180,E1 -19032.789,E2 -19032.789} C_VEL
LIN {X 0,Y 248.986,Z 653.59,A -85,B 0,C 180,E1 -19037.356,E2 -19037.356} C_VEL
LIN {X 0,Y 249.023,Z 653.556,A -85,B 0,C 180,E1 -19042.207,E2 -19042.207} C_VEL
LIN {X 0,Y 249.045,Z 653.58,A -85,B 0,C 180,E1 -19045.639,E2 -19045.639} C_VEL
LIN {X 0,Y 249.005,Z 653.577,A -85,B 0,C 180,E1 -19049.466,E2 -19049.466} C_VEL
LIN {X 0,Y 249.038,Z 653.59,A -85,B 0,C 180,E1 -19053.157,E2 -19053.157} C_VEL
LIN {X 0,Y 249.056,Z 653.571,A -85,B 0,C 180,E1 -19056.73,E2 -19056.73} C_VEL
LIN {X 0,Y 249.088,Z 653.578,A -85,B 0,C 180,E1 -19060.209,E2 -19060.209} C_VEL
LIN {X 0,Y 249.198,Z 653.551,A -85,B 0,C 180,E1 -19063.618,E2 -19063.618} C_VEL
LIN {X 0,Y 249.236,Z 653.547,A -85,B 0,C 180,E1 -19068.615,E2 -19068.615} C_VEL
LIN {X 0,Y 249.438,Z 653.533,A -85,B 0,C 180,E1 -19071.901,E2 -19071.901} C_VEL
LIN {X 0,Y 249.307,Z 653.548,A -85,B 0,C 180,E1 -19074.654,E2 -19074.654} C_VEL
LIN {X 0,Y 248.661,Z 653.63,A -85,B 0,C 180,E1 -19076.005,E2 -19076.005} C_VEL
LIN {X 0,Y 246.088,Z 653.957,A -85,B 0,C 180,E1 -19078.218,E2 -19078.218} C_VEL
LIN {X 0,Y 243.025,Z 654.33,A -85,B 0,C 180,E1 -19080.936,E2 -19080.936} C_VEL
LIN {X 0,Y 242.592,Z 654.382,A -85,B 0,C 180,E1 -19081.872,E2 -19081.872} C_VEL
LIN {X 0,Y 242.425,Z 654.406,A -85,B 0,C 180,E1 -19086.659,E2 -19086.659} C_VEL
LIN {X 0,Y 242.27,Z 654.424,A -85,B 0,C 180,E1 -19090.023,E2 -19090.023} C_VEL
LIN {X 0,Y 242.169,Z 654.434,A -85,B 0,C 180,E1 -19095.14,E2 -19095.14} C_VEL
LIN {X 0,Y 242.075,Z 654.449,A -85,B 0,C 180,E1 -19098.624,E2 -19098.624} C_VEL
LIN {X 0,Y 242.008,Z 654.461,A -85,B 0,C 180,E1 -19102.18,E2 -19102.18} C_VEL
LIN {X 0,Y 242.068,Z 654.456,A -85,B 0,C 180,E1 -19105.838,E2 -19105.838} C_VEL
LIN {X 0,Y 242.032,Z 654.461,A -85,B 0,C 180,E1 -19109.58,E2 -19109.58} C_VEL
LIN {X 0,Y 241.992,Z 654.463,A -85,B 0,C 180,E1 -19113.49,E2 -19113.49} C_VEL
LIN {X 0,Y 242.013,Z 654.462,A -85,B 0,C 180,E1 -19117.577,E2 -19117.577} C_VEL
LIN {X 0,Y 241.963,Z 654.466,A -85,B 0,C 180,E1 -19121.917,E2 -19121.917} C_VEL
LIN {X 0,Y 241.991,Z 654.462,A -85,B 0,C 180,E1 -19125.667,E2 -19125.667} C_VEL
LIN {X 0,Y 244.912,Z 664.92,A -85,B 0,C 180,E1 -19130.06,E2 -19130.06} C_VEL
LIN {X 0,Y 251.917,Z 678.823,A -85,B 0,C 180,E1 -19131.751,E2 -19131.751} C_VEL
LIN {X 0,Y 258.765,Z 694.124,A -85,B 0,C 180,E1 -19133.341,E2 -19133.341} C_VEL
LIN {X 0,Y 263.583,Z 706.366,A -85,B 0,C 180,E1 -19134.442,E2 -19134.442} C_VEL
LIN {X 0,Y 265.916,Z 724.945,A -85,B 0,C 180,E1 -19135.352,E2 -19135.352} C_VEL
LIN {X 0,Y 262.715,Z 803.646,A -85,B 0,C 180,E1 -19137.427,E2 -19137.427} C_VEL
LIN {X 0,Y 261.363,Z 818.366,A -85,B 0,C 180,E1 -19138.092,E2 -19138.092} C_VEL
LIN {X 0,Y 259.576,Z 832.409,A -85,B 0,C 180,E1 -19139.041,E2 -19139.041} C_VEL
LIN {X 0,Y 257.553,Z 844.557,A -85,B 0,C 180,E1 -19140.132,E2 -19140.132} C_VEL
LIN {X 0,Y 255.107,Z 857.382,A -85,B 0,C 180,E1 -19141.626,E2 -19141.626} C_VEL
LIN {X 0,Y 252.728,Z 868.487,A -85,B 0,C 180,E1 -19143.251,E2 -19143.251} C_VEL
LIN {X 0,Y 250.295,Z 878.761,A -85,B 0,C 180,E1 -19145.09,E2 -19145.09} C_VEL
LIN {X 0,Y 247.948,Z 887.882,A -85,B 0,C 180,E1 -19147.061,E2 -19147.061} C_VEL
LIN {X 0,Y 245.665,Z 897.052,A -85,B 0,C 180,E1 -19149.485,E2 -19149.485} C_VEL
LIN {X 0,Y 243.453,Z 905.658,A -85,B 0,C 180,E1 -19152.296,E2 -19152.296} C_VEL
LIN {X 0,Y 242.117,Z 911.977,A -85,B 0,C 180,E1 -19154.856,E2 -19154.856} C_VEL
LIN {X 0,Y 241.029,Z 917.074,A -85,B 0,C 180,E1 -19157.368,E2 -19157.368} C_VEL
LIN {X 0,Y 240.208,Z 922.323,A -85,B 0,C 180,E1 -19160.74,E2 -19160.74} C_VEL
LIN {X 0,Y 239.915,Z 925.27,A -85,B 0,C 180,E1 -19163.271,E2 -19163.271} C_VEL
LIN {X 0,Y 239.899,Z 926.774,A -85,B 0,C 180,E1 -19164.958,E2 -19164.958} C_VEL
LIN {X 0,Y 239.919,Z 928.714,A -85,B 0,C 180,E1 -19168.321,E2 -19168.321} C_VEL
LIN {X 0,Y 239.958,Z 929.167,A -85,B 0,C 180,E1 -19170,E2 -19170} C_VEL
LIN {X 0,Y 239.908,Z 929.277,A -85,B 0,C 180,E1 -19171.679,E2 -19171.679} C_VEL
LIN {X 0,Y 239.843,Z 928.49,A -85,B 0,C 180,E1 -19175.043,E2 -19175.043} C_VEL
